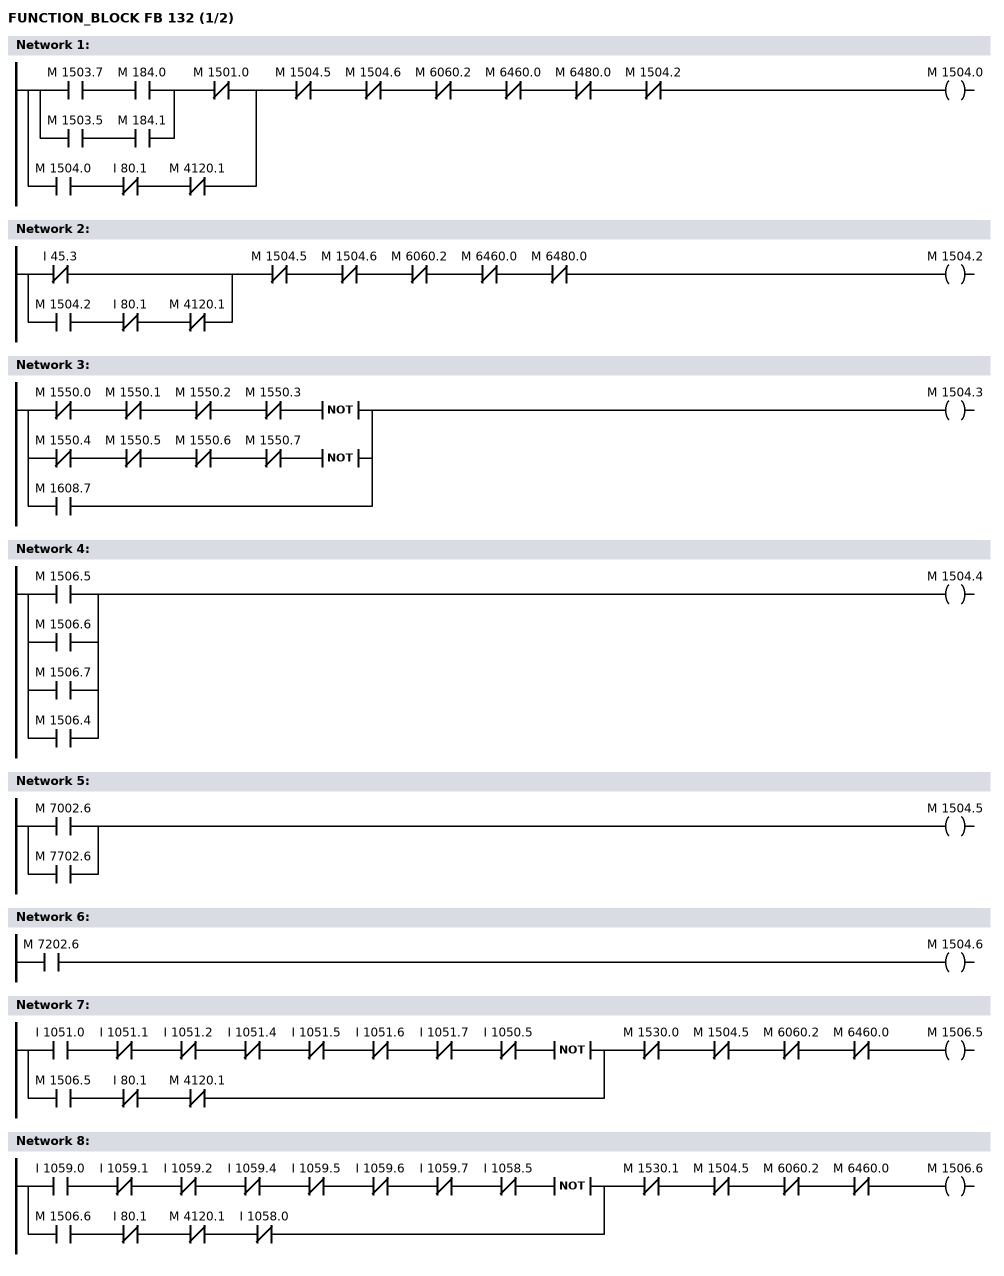

      A(    ;
      A(    ;
      A     M   1503.7;
      A     M    184.0;
      O     ;
      A     M   1503.5;
      A     M    184.1;
      )     ;
      AN    M   1501.0;
      O     ;
      A     M   1504.0;
      AN    I     80.1;
      AN    M   4120.1;
      )     ;
      AN    M   1504.5;
      AN    M   1504.6;
      AN    M   6060.2;
      AN    M   6460.0;
      AN    M   6480.0;
      AN    M   1504.2;
      =     M   1504.0;
NETWORK
TITLE =

      A(    ;
      ON    I     45.3;
      O     ;
      A     M   1504.2;
      AN    I     80.1;
      AN    M   4120.1;
      )     ;
      AN    M   1504.5;
      AN    M   1504.6;
      AN    M   6060.2;
      AN    M   6460.0;
      AN    M   6480.0;
      =     M   1504.2;
NETWORK
TITLE =

      AN    M   1550.0;
      AN    M   1550.1;
      AN    M   1550.2;
      AN    M   1550.3;
      NOT   ;
      O(    ;
      AN    M   1550.4;
      AN    M   1550.5;
      AN    M   1550.6;
      AN    M   1550.7;
      NOT   ;
      )     ;
      O     M   1608.7;
      =     M   1504.3;
NETWORK
TITLE =

      O     M   1506.5;
      O     M   1506.6;
      O     M   1506.7;
      O     M   1506.4;
      =     M   1504.4;
NETWORK
TITLE =

      O     M   7002.6;
      O     M   7702.6;
      =     M   1504.5;
NETWORK
TITLE =

      A     M   7202.6;
      =     M   1504.6;
NETWORK
TITLE =

      A(    ;
      A     I   1051.0;
      AN    I   1051.1;
      AN    I   1051.2;
      AN    I   1051.4;
      AN    I   1051.5;
      AN    I   1051.6;
      AN    I   1051.7;
      AN    I   1050.5;
      NOT   ;
      O     ;
      A     M   1506.5;
      AN    I     80.1;
      AN    M   4120.1;
      )     ;
      AN    M   1530.0;
      AN    M   1504.5;
      AN    M   6060.2;
      AN    M   6460.0;
      =     M   1506.5;
NETWORK
TITLE =

      A(    ;
      A     I   1059.0;
      AN    I   1059.1;
      AN    I   1059.2;
      AN    I   1059.4;
      AN    I   1059.5;
      AN    I   1059.6;
      AN    I   1059.7;
      AN    I   1058.5;
      NOT   ;
      O     ;
      A     M   1506.6;
      AN    I     80.1;
      AN    M   4120.1;
      AN    I   1058.0;
      )     ;
      AN    M   1530.1;
      AN    M   1504.5;
      AN    M   6060.2;
      AN    M   6460.0;
      =     M   1506.6;
NETWORK
TITLE =
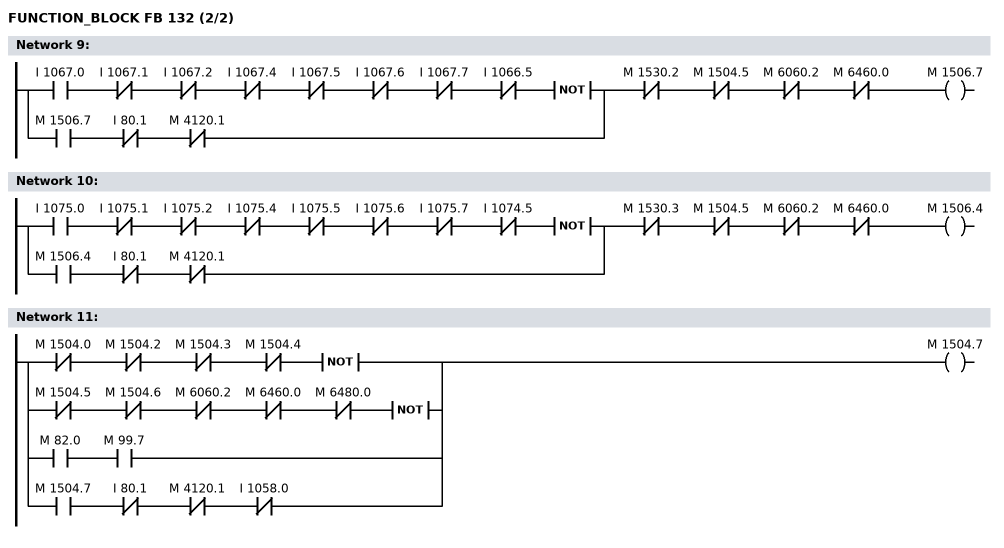

      A(    ;
      A     I   1067.0;
      AN    I   1067.1;
      AN    I   1067.2;
      AN    I   1067.4;
      AN    I   1067.5;
      AN    I   1067.6;
      AN    I   1067.7;
      AN    I   1066.5;
      NOT   ;
      O     ;
      A     M   1506.7;
      AN    I     80.1;
      AN    M   4120.1;
      )     ;
      AN    M   1530.2;
      AN    M   1504.5;
      AN    M   6060.2;
      AN    M   6460.0;
      =     M   1506.7;
NETWORK
TITLE =

      A(    ;
      A     I   1075.0;
      AN    I   1075.1;
      AN    I   1075.2;
      AN    I   1075.4;
      AN    I   1075.5;
      AN    I   1075.6;
      AN    I   1075.7;
      AN    I   1074.5;
      NOT   ;
      O     ;
      A     M   1506.4;
      AN    I     80.1;
      AN    M   4120.1;
      )     ;
      AN    M   1530.3;
      AN    M   1504.5;
      AN    M   6060.2;
      AN    M   6460.0;
      =     M   1506.4;
NETWORK
TITLE =

      AN    M   1504.0;
      AN    M   1504.2;
      AN    M   1504.3;
      AN    M   1504.4;
      NOT   ;
      O(    ;
      AN    M   1504.5;
      AN    M   1504.6;
      AN    M   6060.2;
      AN    M   6460.0;
      AN    M   6480.0;
      NOT   ;
      )     ;
      O     ;
      A     M     82.0;
      A     M     99.7;
      O     ;
      A     M   1504.7;
      AN    I     80.1;
      AN    M   4120.1;
      AN    I   1058.0;
      =     M   1504.7;
END_FUNCTION_BLOCK

DATA_BLOCK DB 132
TITLE =
VERSION : 0.0

 FB 132
BEGIN
END_DATA_BLOCK

FUNCTION FC 132 : VOID
TITLE =
VERSION : 0.1

BEGIN
NETWORK
TITLE =
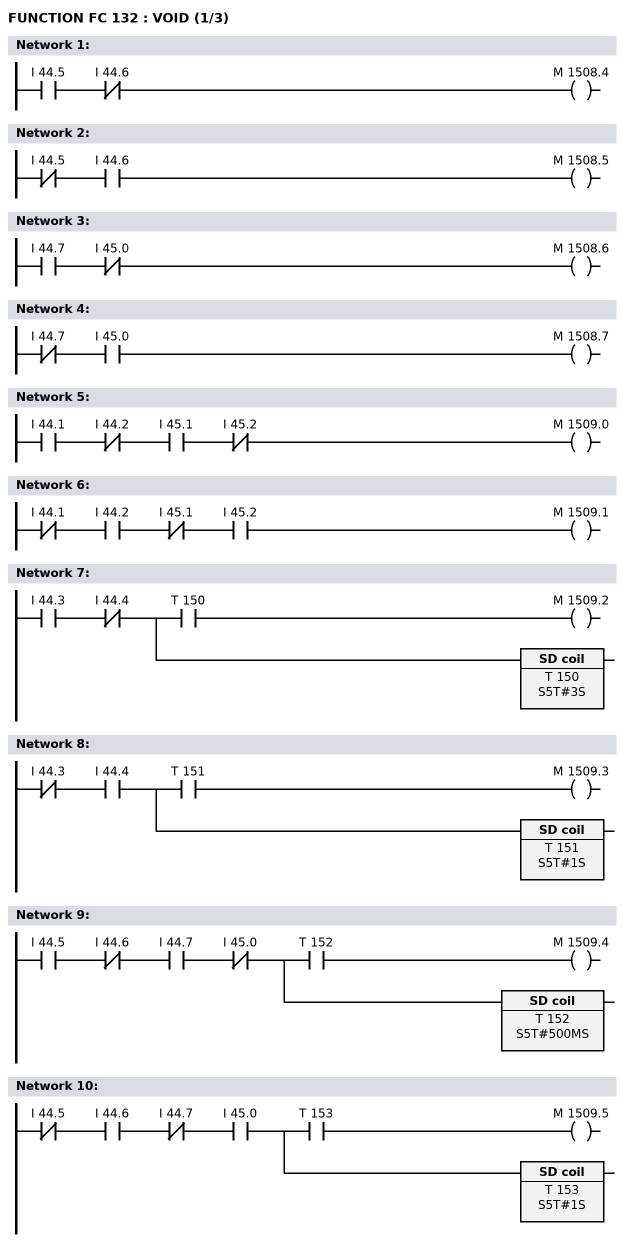

      A     I     44.5;
      AN    I     44.6;
      =     M   1508.4;
NETWORK
TITLE =

      AN    I     44.5;
      A     I     44.6;
      =     M   1508.5;
NETWORK
TITLE =

      A     I     44.7;
      AN    I     45.0;
      =     M   1508.6;
NETWORK
TITLE =

      AN    I     44.7;
      A     I     45.0;
      =     M   1508.7;
NETWORK
TITLE =

      A     I     44.1;
      AN    I     44.2;
      A     I     45.1;
      AN    I     45.2;
      =     M   1509.0;
NETWORK
TITLE =

      AN    I     44.1;
      A     I     44.2;
      AN    I     45.1;
      A     I     45.2;
      =     M   1509.1;
NETWORK
TITLE =

      A     I     44.3;
      AN    I     44.4;
      =     L      0.0;
      A     L      0.0;
      A     T    150;
      =     M   1509.2;
      A     L      0.0;
      BLD   102;
      L     S5T#3S;
      SD    T    150;
NETWORK
TITLE =

      AN    I     44.3;
      A     I     44.4;
      =     L      0.0;
      A     L      0.0;
      A     T    151;
      =     M   1509.3;
      A     L      0.0;
      BLD   102;
      L     S5T#1S;
      SD    T    151;
NETWORK
TITLE =

      A     I     44.5;
      AN    I     44.6;
      A     I     44.7;
      AN    I     45.0;
      =     L      0.0;
      A     L      0.0;
      A     T    152;
      =     M   1509.4;
      A     L      0.0;
      BLD   102;
      L     S5T#500MS;
      SD    T    152;
NETWORK
TITLE =

      AN    I     44.5;
      A     I     44.6;
      AN    I     44.7;
      A     I     45.0;
      =     L      0.0;
      A     L      0.0;
      A     T    153;
      =     M   1509.5;
      A     L      0.0;
      BLD   102;
      L     S5T#1S;
      SD    T    153;
NETWORK
TITLE =
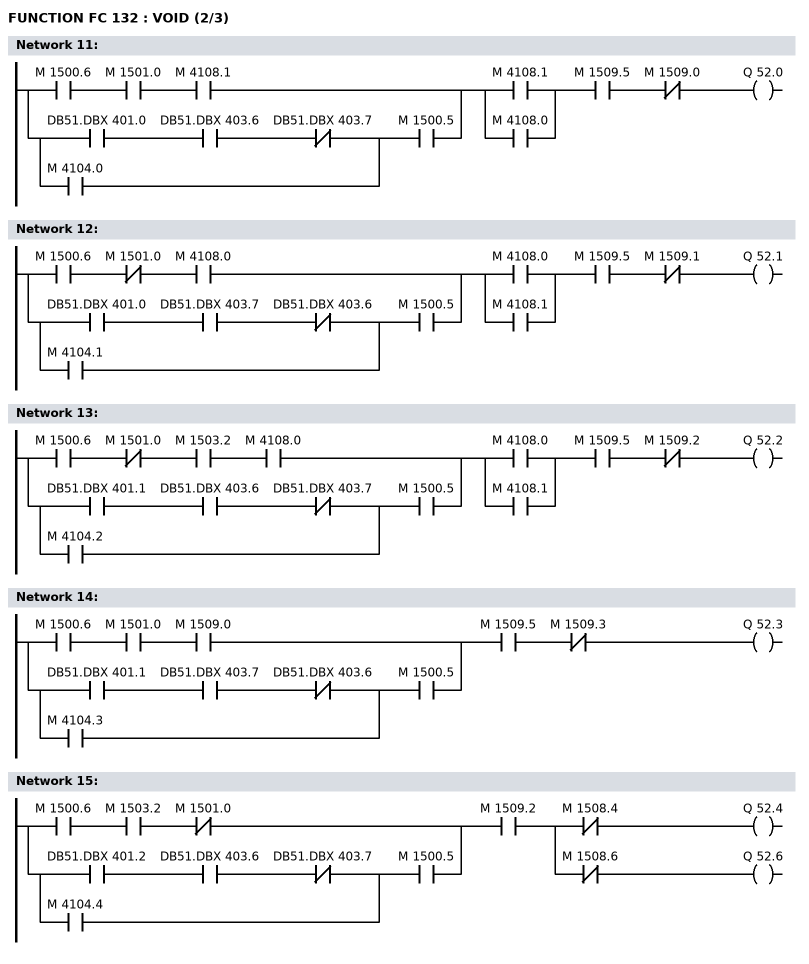

      A(    ;
      A     M   1500.6;
      A     M   1501.0;
      A     M   4108.1;
      O     ;
      A(    ;
      A     DB51.DBX  401.0;
      A     DB51.DBX  403.6;
      AN    DB51.DBX  403.7;
      O     M   4104.0;
      )     ;
      A     M   1500.5;
      )     ;
      A(    ;
      O     M   4108.1;
      O     M   4108.0;
      )     ;
      A     M   1509.5;
      AN    M   1509.0;
      =     Q     52.0;
NETWORK
TITLE =

      A(    ;
      A     M   1500.6;
      AN    M   1501.0;
      A     M   4108.0;
      O     ;
      A(    ;
      A     DB51.DBX  401.0;
      A     DB51.DBX  403.7;
      AN    DB51.DBX  403.6;
      O     M   4104.1;
      )     ;
      A     M   1500.5;
      )     ;
      A(    ;
      O     M   4108.0;
      O     M   4108.1;
      )     ;
      A     M   1509.5;
      AN    M   1509.1;
      =     Q     52.1;
NETWORK
TITLE =

      A(    ;
      A     M   1500.6;
      AN    M   1501.0;
      A     M   1503.2;
      A     M   4108.0;
      O     ;
      A(    ;
      A     DB51.DBX  401.1;
      A     DB51.DBX  403.6;
      AN    DB51.DBX  403.7;
      O     M   4104.2;
      )     ;
      A     M   1500.5;
      )     ;
      A(    ;
      O     M   4108.0;
      O     M   4108.1;
      )     ;
      A     M   1509.5;
      AN    M   1509.2;
      =     Q     52.2;
NETWORK
TITLE =

      A(    ;
      A     M   1500.6;
      A     M   1501.0;
      A     M   1509.0;
      O     ;
      A(    ;
      A     DB51.DBX  401.1;
      A     DB51.DBX  403.7;
      AN    DB51.DBX  403.6;
      O     M   4104.3;
      )     ;
      A     M   1500.5;
      )     ;
      A     M   1509.5;
      AN    M   1509.3;
      =     Q     52.3;
NETWORK
TITLE =

      A(    ;
      A     M   1500.6;
      A     M   1503.2;
      AN    M   1501.0;
      O     ;
      A(    ;
      A     DB51.DBX  401.2;
      A     DB51.DBX  403.6;
      AN    DB51.DBX  403.7;
      O     M   4104.4;
      )     ;
      A     M   1500.5;
      )     ;
      A     M   1509.2;
      =     L      0.0;
      A     L      0.0;
      AN    M   1508.4;
      =     Q     52.4;
      A     L      0.0;
      AN    M   1508.6;
      =     Q     52.6;
NETWORK
TITLE =
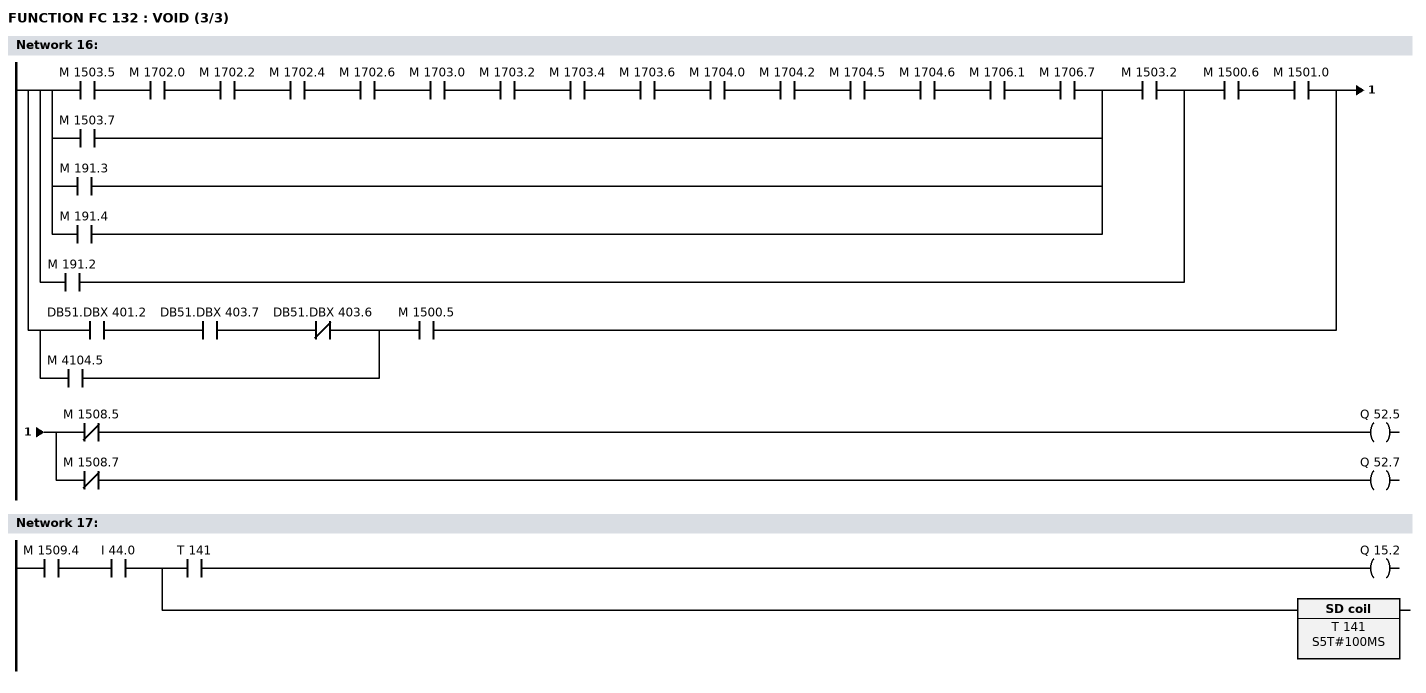

      A(    ;
      A(    ;
      A     M   1503.5;
      A     M   1702.0;
      A     M   1702.2;
      A     M   1702.4;
      A     M   1702.6;
      A     M   1703.0;
      A     M   1703.2;
      A     M   1703.4;
      A     M   1703.6;
      A     M   1704.0;
      A     M   1704.2;
      A     M   1704.5;
      A     M   1704.6;
      A     M   1706.1;
      A     M   1706.7;
      O     M   1503.7;
      O     M    191.3;
      O     M    191.4;
      )     ;
      A     M   1503.2;
      O     M    191.2;
      )     ;
      A     M   1500.6;
      A     M   1501.0;
      O     ;
      A(    ;
      A     DB51.DBX  401.2;
      A     DB51.DBX  403.7;
      AN    DB51.DBX  403.6;
      O     M   4104.5;
      )     ;
      A     M   1500.5;
      =     L      0.0;
      A     L      0.0;
      AN    M   1508.5;
      =     Q     52.5;
      A     L      0.0;
      AN    M   1508.7;
      =     Q     52.7;
NETWORK
TITLE =

      A     M   1509.4;
      A     I     44.0;
      =     L      0.0;
      A     L      0.0;
      A     T    141;
      =     Q     15.2;
      A     L      0.0;
      BLD   102;
      L     S5T#100MS;
      SD    T    141;
END_FUNCTION

FUNCTION_BLOCK FB 133
TITLE =
VERSION : 0.1


VAR
  S707_LM_DC_PIN : FB 424;
  S707_LM_DC_1ST_CLAMP1 : FB 424;
  S707_LM_DC_1ST_CLAMP2 : FB 424;
  S707_LM_DC_1ST_CLAMP3 : FB 424;
  S707_LM_DC_1ST_CLAMP4 : FB 424;
  S707_LM_DC_2ND_CLAMP1 : FB 424;
  S707_LM_DC_2ND_CLAMP2 : FB 424;
  S707_LM_DC_2ND_CLAMP3 : FB 424;
  S707_LM_DC_2ND_CLAMP4 : FB 424;
  S707_LM_DC_2ND_CLAMP5 : FB 424;
  S707_LM_DC_STK_PIN : FB 424;
  S707_LM_DC_OTR_CLAMP : FB 424;
  S707_LM_DC_ASSY_CLAMP : FB 424;
  S707_LM_DC_FF_PIN : FB 424;
  S707_LM_DC_FF_CLAMP : FB 424;
  S707_LM_DC_2ND_CLAMP6 : FB 424;
  S707_LM_DC_2ND_CLAMP7 : FB 424;
  S707_LM_DC_1ST_CLAMP5 : FB 424;
END_VAR
BEGIN
NETWORK
TITLE =
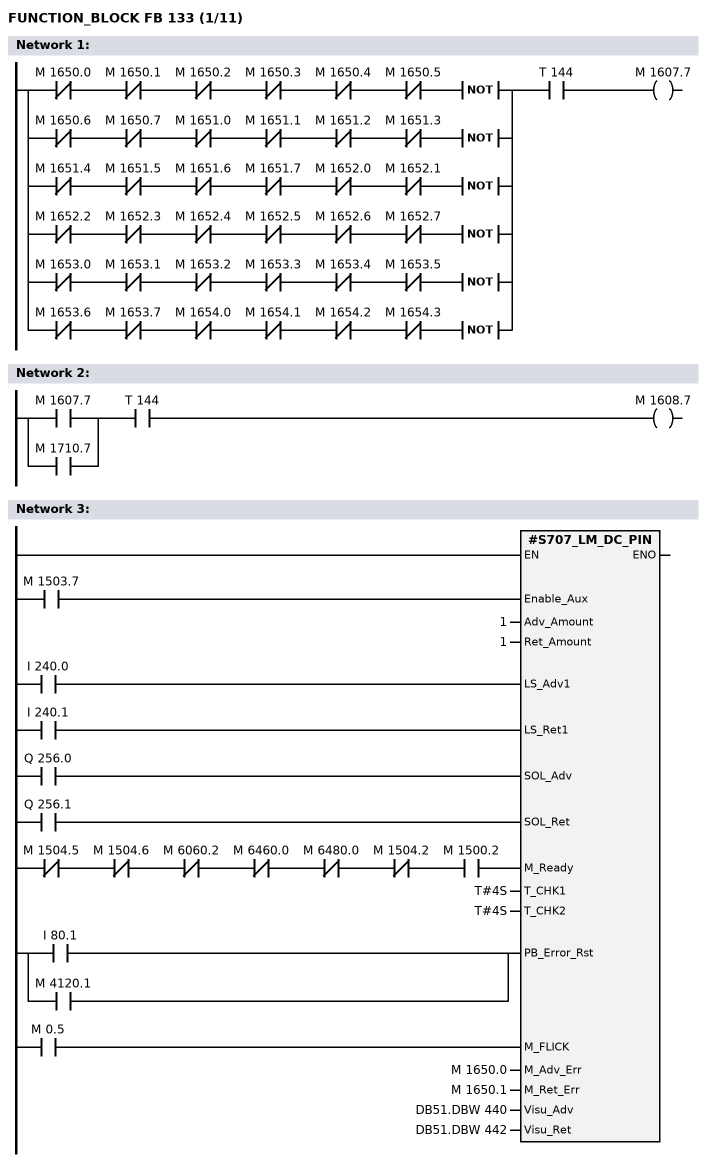

      A(    ;
      AN    M   1650.0;
      AN    M   1650.1;
      AN    M   1650.2;
      AN    M   1650.3;
      AN    M   1650.4;
      AN    M   1650.5;
      NOT   ;
      O(    ;
      AN    M   1650.6;
      AN    M   1650.7;
      AN    M   1651.0;
      AN    M   1651.1;
      AN    M   1651.2;
      AN    M   1651.3;
      NOT   ;
      )     ;
      O(    ;
      AN    M   1651.4;
      AN    M   1651.5;
      AN    M   1651.6;
      AN    M   1651.7;
      AN    M   1652.0;
      AN    M   1652.1;
      NOT   ;
      )     ;
      O(    ;
      AN    M   1652.2;
      AN    M   1652.3;
      AN    M   1652.4;
      AN    M   1652.5;
      AN    M   1652.6;
      AN    M   1652.7;
      NOT   ;
      )     ;
      O(    ;
      AN    M   1653.0;
      AN    M   1653.1;
      AN    M   1653.2;
      AN    M   1653.3;
      AN    M   1653.4;
      AN    M   1653.5;
      NOT   ;
      )     ;
      O(    ;
      AN    M   1653.6;
      AN    M   1653.7;
      AN    M   1654.0;
      AN    M   1654.1;
      AN    M   1654.2;
      AN    M   1654.3;
      NOT   ;
      )     ;
      )     ;
      A     T    144;
      =     M   1607.7;
NETWORK
TITLE =

      A(    ;
      O     M   1607.7;
      O     M   1710.7;
      )     ;
      A     T    144;
      =     M   1608.7;
NETWORK
TITLE =

      A     M   1503.7;
      =     L      0.0;
      BLD   103;
      A     I    240.0;
      =     L      0.1;
      BLD   103;
      A     I    240.1;
      =     L      0.2;
      BLD   103;
      A     Q    256.0;
      =     L      1.1;
      BLD   103;
      A     Q    256.1;
      =     L      1.2;
      BLD   103;
      AN    M   1504.5;
      AN    M   1504.6;
      AN    M   6060.2;
      AN    M   6460.0;
      AN    M   6480.0;
      AN    M   1504.2;
      A     M   1500.2;
      =     L      1.3;
      BLD   103;
      A(    ;
      O     I     80.1;
      O     M   4120.1;
      )     ;
      =     L      1.5;
      BLD   103;
      A     M      0.5;
      =     L      1.6;
      BLD   103;
      CALL #S707_LM_DC_PIN (
           Enable_Aux               := L      0.0,
           Adv_Amount               := 1,
           Ret_Amount               := 1,
           LS_Adv1                  := L      0.1,
           LS_Ret1                  := L      0.2,
           SOL_Adv                  := L      1.1,
           SOL_Ret                  := L      1.2,
           M_Ready                  := L      1.3,
           T_CHK1                   := T#4S,
           T_CHK2                   := T#4S,
           PB_Error_Rst             := L      1.5,
           M_FLICK                  := L      1.6,
           M_Adv_Err                := M   1650.0,
           M_Ret_Err                := M   1650.1,
           Visu_Adv                 := DB51.DBW  440,
           Visu_Ret                 := DB51.DBW  442);
      NOP   0;
NETWORK
TITLE =
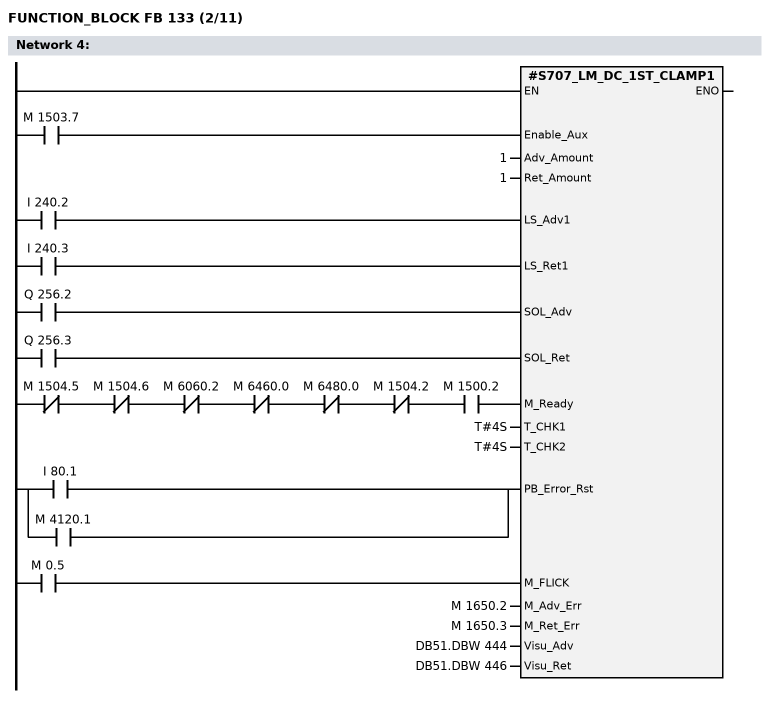

      A     M   1503.7;
      =     L      0.0;
      BLD   103;
      A     I    240.2;
      =     L      0.1;
      BLD   103;
      A     I    240.3;
      =     L      0.2;
      BLD   103;
      A     Q    256.2;
      =     L      1.1;
      BLD   103;
      A     Q    256.3;
      =     L      1.2;
      BLD   103;
      AN    M   1504.5;
      AN    M   1504.6;
      AN    M   6060.2;
      AN    M   6460.0;
      AN    M   6480.0;
      AN    M   1504.2;
      A     M   1500.2;
      =     L      1.3;
      BLD   103;
      A(    ;
      O     I     80.1;
      O     M   4120.1;
      )     ;
      =     L      1.5;
      BLD   103;
      A     M      0.5;
      =     L      1.6;
      BLD   103;
      CALL #S707_LM_DC_1ST_CLAMP1 (
           Enable_Aux               := L      0.0,
           Adv_Amount               := 1,
           Ret_Amount               := 1,
           LS_Adv1                  := L      0.1,
           LS_Ret1                  := L      0.2,
           SOL_Adv                  := L      1.1,
           SOL_Ret                  := L      1.2,
           M_Ready                  := L      1.3,
           T_CHK1                   := T#4S,
           T_CHK2                   := T#4S,
           PB_Error_Rst             := L      1.5,
           M_FLICK                  := L      1.6,
           M_Adv_Err                := M   1650.2,
           M_Ret_Err                := M   1650.3,
           Visu_Adv                 := DB51.DBW  444,
           Visu_Ret                 := DB51.DBW  446);
      NOP   0;
NETWORK
TITLE =
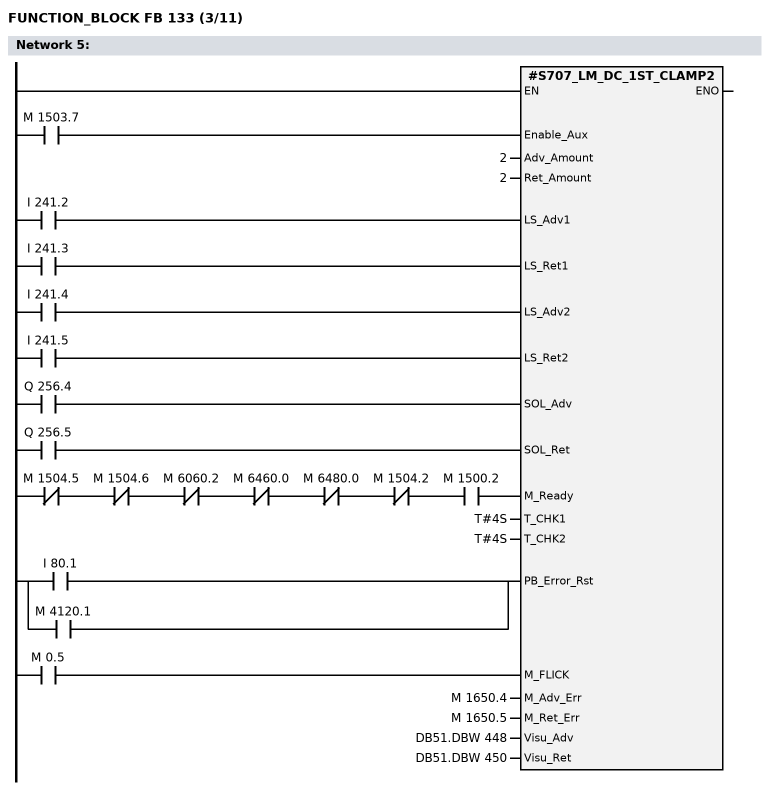

      A     M   1503.7;
      =     L      0.0;
      BLD   103;
      A     I    241.2;
      =     L      0.1;
      BLD   103;
      A     I    241.3;
      =     L      0.2;
      BLD   103;
      A     I    241.4;
      =     L      0.3;
      BLD   103;
      A     I    241.5;
      =     L      0.4;
      BLD   103;
      A     Q    256.4;
      =     L      1.1;
      BLD   103;
      A     Q    256.5;
      =     L      1.2;
      BLD   103;
      AN    M   1504.5;
      AN    M   1504.6;
      AN    M   6060.2;
      AN    M   6460.0;
      AN    M   6480.0;
      AN    M   1504.2;
      A     M   1500.2;
      =     L      1.3;
      BLD   103;
      A(    ;
      O     I     80.1;
      O     M   4120.1;
      )     ;
      =     L      1.5;
      BLD   103;
      A     M      0.5;
      =     L      1.6;
      BLD   103;
      CALL #S707_LM_DC_1ST_CLAMP2 (
           Enable_Aux               := L      0.0,
           Adv_Amount               := 2,
           Ret_Amount               := 2,
           LS_Adv1                  := L      0.1,
           LS_Ret1                  := L      0.2,
           LS_Adv2                  := L      0.3,
           LS_Ret2                  := L      0.4,
           SOL_Adv                  := L      1.1,
           SOL_Ret                  := L      1.2,
           M_Ready                  := L      1.3,
           T_CHK1                   := T#4S,
           T_CHK2                   := T#4S,
           PB_Error_Rst             := L      1.5,
           M_FLICK                  := L      1.6,
           M_Adv_Err                := M   1650.4,
           M_Ret_Err                := M   1650.5,
           Visu_Adv                 := DB51.DBW  448,
           Visu_Ret                 := DB51.DBW  450);
      NOP   0;
NETWORK
TITLE =
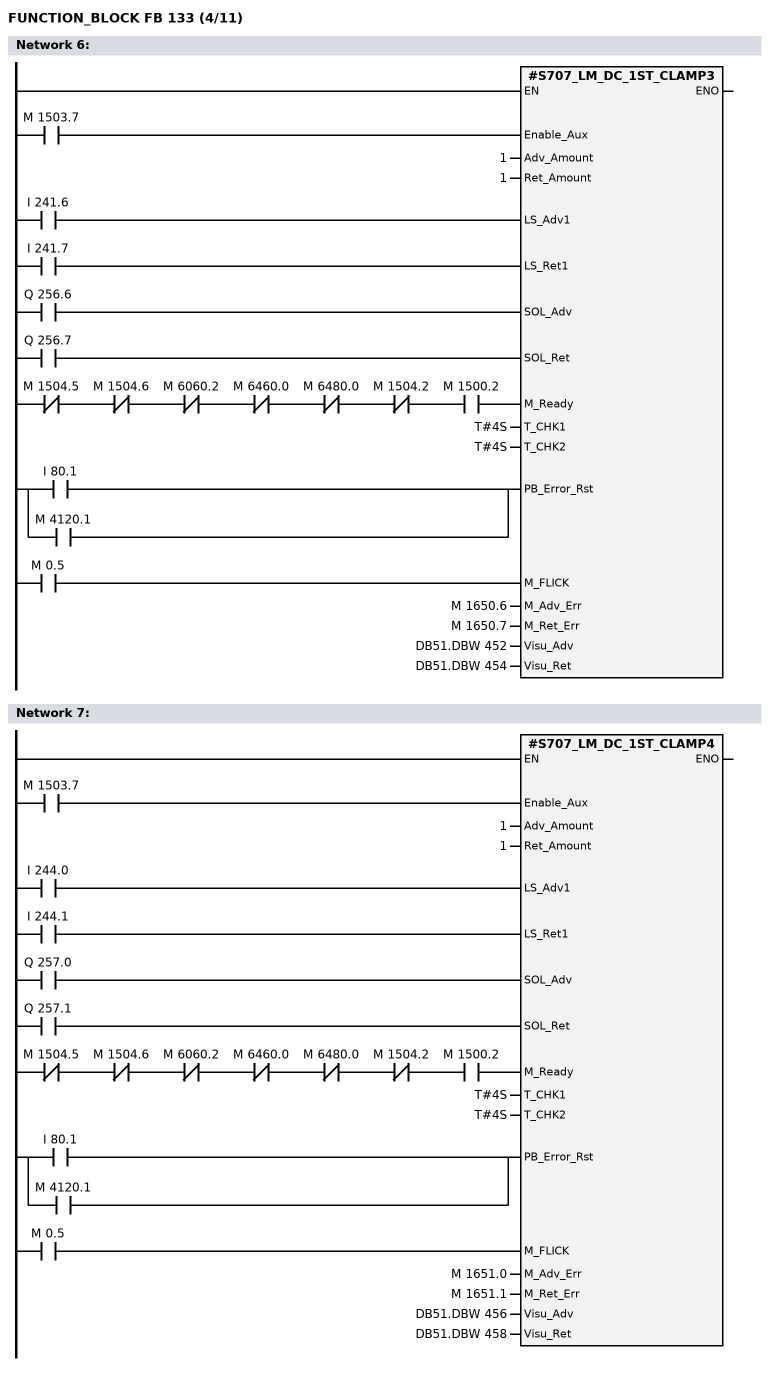

      A     M   1503.7;
      =     L      0.0;
      BLD   103;
      A     I    241.6;
      =     L      0.1;
      BLD   103;
      A     I    241.7;
      =     L      0.2;
      BLD   103;
      A     Q    256.6;
      =     L      1.1;
      BLD   103;
      A     Q    256.7;
      =     L      1.2;
      BLD   103;
      AN    M   1504.5;
      AN    M   1504.6;
      AN    M   6060.2;
      AN    M   6460.0;
      AN    M   6480.0;
      AN    M   1504.2;
      A     M   1500.2;
      =     L      1.3;
      BLD   103;
      A(    ;
      O     I     80.1;
      O     M   4120.1;
      )     ;
      =     L      1.5;
      BLD   103;
      A     M      0.5;
      =     L      1.6;
      BLD   103;
      CALL #S707_LM_DC_1ST_CLAMP3 (
           Enable_Aux               := L      0.0,
           Adv_Amount               := 1,
           Ret_Amount               := 1,
           LS_Adv1                  := L      0.1,
           LS_Ret1                  := L      0.2,
           SOL_Adv                  := L      1.1,
           SOL_Ret                  := L      1.2,
           M_Ready                  := L      1.3,
           T_CHK1                   := T#4S,
           T_CHK2                   := T#4S,
           PB_Error_Rst             := L      1.5,
           M_FLICK                  := L      1.6,
           M_Adv_Err                := M   1650.6,
           M_Ret_Err                := M   1650.7,
           Visu_Adv                 := DB51.DBW  452,
           Visu_Ret                 := DB51.DBW  454);
      NOP   0;
NETWORK
TITLE =

      A     M   1503.7;
      =     L      0.0;
      BLD   103;
      A     I    244.0;
      =     L      0.1;
      BLD   103;
      A     I    244.1;
      =     L      0.2;
      BLD   103;
      A     Q    257.0;
      =     L      1.1;
      BLD   103;
      A     Q    257.1;
      =     L      1.2;
      BLD   103;
      AN    M   1504.5;
      AN    M   1504.6;
      AN    M   6060.2;
      AN    M   6460.0;
      AN    M   6480.0;
      AN    M   1504.2;
      A     M   1500.2;
      =     L      1.3;
      BLD   103;
      A(    ;
      O     I     80.1;
      O     M   4120.1;
      )     ;
      =     L      1.5;
      BLD   103;
      A     M      0.5;
      =     L      1.6;
      BLD   103;
      CALL #S707_LM_DC_1ST_CLAMP4 (
           Enable_Aux               := L      0.0,
           Adv_Amount               := 1,
           Ret_Amount               := 1,
           LS_Adv1                  := L      0.1,
           LS_Ret1                  := L      0.2,
           SOL_Adv                  := L      1.1,
           SOL_Ret                  := L      1.2,
           M_Ready                  := L      1.3,
           T_CHK1                   := T#4S,
           T_CHK2                   := T#4S,
           PB_Error_Rst             := L      1.5,
           M_FLICK                  := L      1.6,
           M_Adv_Err                := M   1651.0,
           M_Ret_Err                := M   1651.1,
           Visu_Adv                 := DB51.DBW  456,
           Visu_Ret                 := DB51.DBW  458);
      NOP   0;
NETWORK
TITLE =
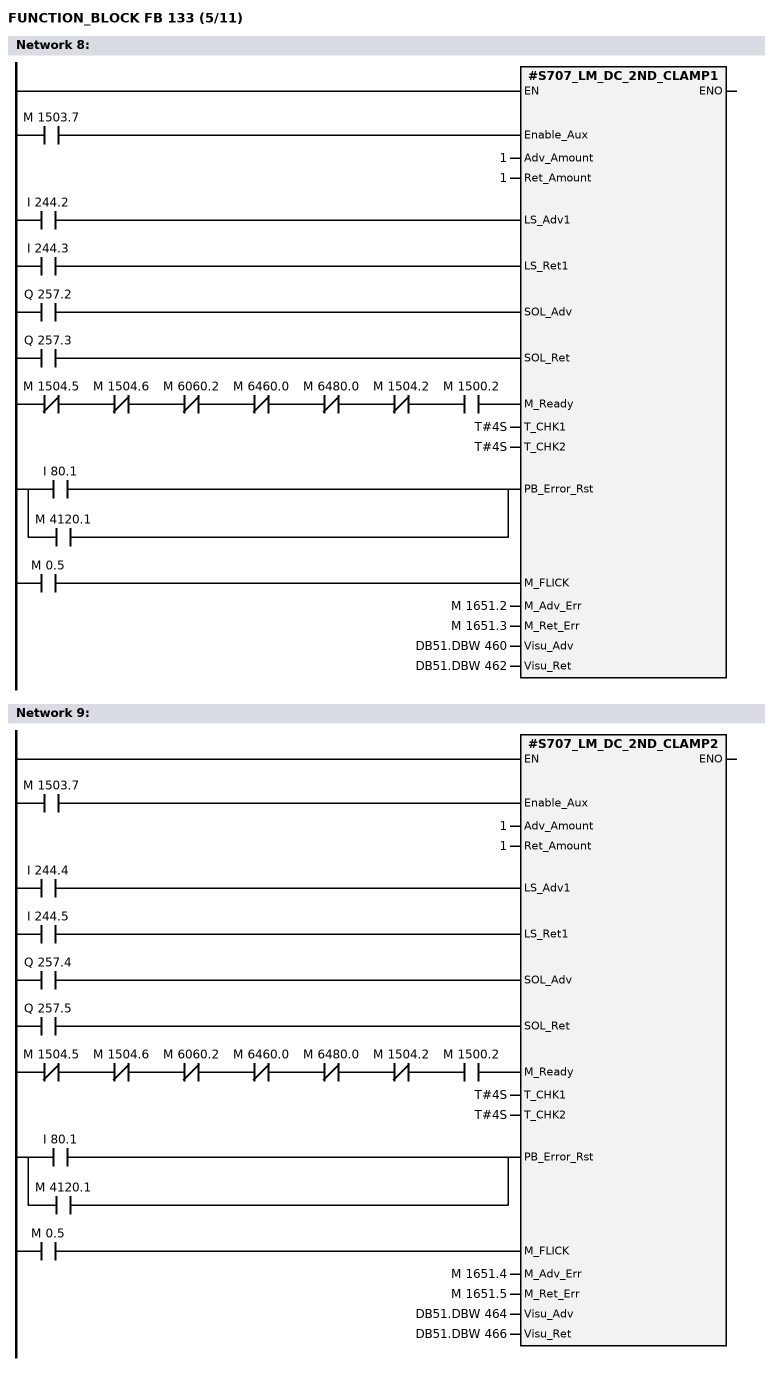

      A     M   1503.7;
      =     L      0.0;
      BLD   103;
      A     I    244.2;
      =     L      0.1;
      BLD   103;
      A     I    244.3;
      =     L      0.2;
      BLD   103;
      A     Q    257.2;
      =     L      1.1;
      BLD   103;
      A     Q    257.3;
      =     L      1.2;
      BLD   103;
      AN    M   1504.5;
      AN    M   1504.6;
      AN    M   6060.2;
      AN    M   6460.0;
      AN    M   6480.0;
      AN    M   1504.2;
      A     M   1500.2;
      =     L      1.3;
      BLD   103;
      A(    ;
      O     I     80.1;
      O     M   4120.1;
      )     ;
      =     L      1.5;
      BLD   103;
      A     M      0.5;
      =     L      1.6;
      BLD   103;
      CALL #S707_LM_DC_2ND_CLAMP1 (
           Enable_Aux               := L      0.0,
           Adv_Amount               := 1,
           Ret_Amount               := 1,
           LS_Adv1                  := L      0.1,
           LS_Ret1                  := L      0.2,
           SOL_Adv                  := L      1.1,
           SOL_Ret                  := L      1.2,
           M_Ready                  := L      1.3,
           T_CHK1                   := T#4S,
           T_CHK2                   := T#4S,
           PB_Error_Rst             := L      1.5,
           M_FLICK                  := L      1.6,
           M_Adv_Err                := M   1651.2,
           M_Ret_Err                := M   1651.3,
           Visu_Adv                 := DB51.DBW  460,
           Visu_Ret                 := DB51.DBW  462);
      NOP   0;
NETWORK
TITLE =

      A     M   1503.7;
      =     L      0.0;
      BLD   103;
      A     I    244.4;
      =     L      0.1;
      BLD   103;
      A     I    244.5;
      =     L      0.2;
      BLD   103;
      A     Q    257.4;
      =     L      1.1;
      BLD   103;
      A     Q    257.5;
      =     L      1.2;
      BLD   103;
      AN    M   1504.5;
      AN    M   1504.6;
      AN    M   6060.2;
      AN    M   6460.0;
      AN    M   6480.0;
      AN    M   1504.2;
      A     M   1500.2;
      =     L      1.3;
      BLD   103;
      A(    ;
      O     I     80.1;
      O     M   4120.1;
      )     ;
      =     L      1.5;
      BLD   103;
      A     M      0.5;
      =     L      1.6;
      BLD   103;
      CALL #S707_LM_DC_2ND_CLAMP2 (
           Enable_Aux               := L      0.0,
           Adv_Amount               := 1,
           Ret_Amount               := 1,
           LS_Adv1                  := L      0.1,
           LS_Ret1                  := L      0.2,
           SOL_Adv                  := L      1.1,
           SOL_Ret                  := L      1.2,
           M_Ready                  := L      1.3,
           T_CHK1                   := T#4S,
           T_CHK2                   := T#4S,
           PB_Error_Rst             := L      1.5,
           M_FLICK                  := L      1.6,
           M_Adv_Err                := M   1651.4,
           M_Ret_Err                := M   1651.5,
           Visu_Adv                 := DB51.DBW  464,
           Visu_Ret                 := DB51.DBW  466);
      NOP   0;
NETWORK
TITLE =
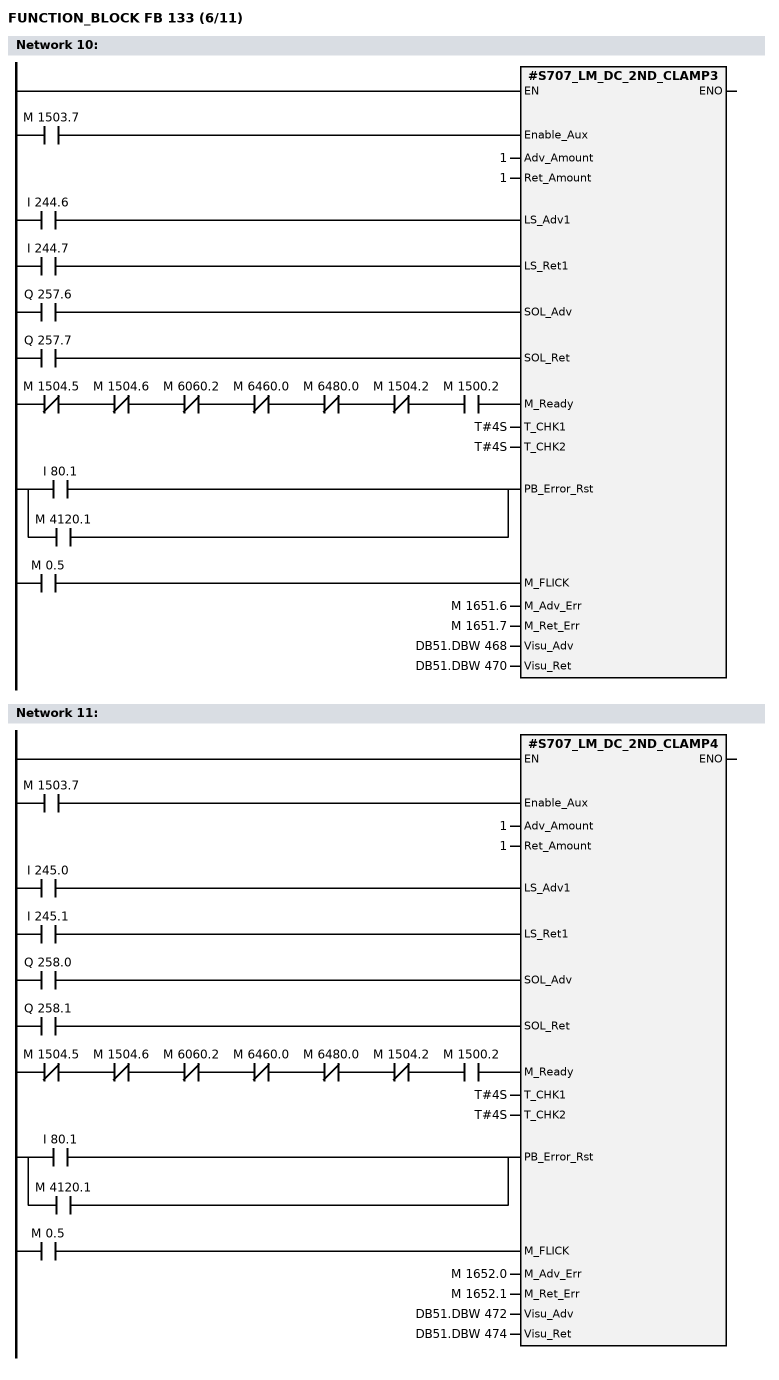

      A     M   1503.7;
      =     L      0.0;
      BLD   103;
      A     I    244.6;
      =     L      0.1;
      BLD   103;
      A     I    244.7;
      =     L      0.2;
      BLD   103;
      A     Q    257.6;
      =     L      1.1;
      BLD   103;
      A     Q    257.7;
      =     L      1.2;
      BLD   103;
      AN    M   1504.5;
      AN    M   1504.6;
      AN    M   6060.2;
      AN    M   6460.0;
      AN    M   6480.0;
      AN    M   1504.2;
      A     M   1500.2;
      =     L      1.3;
      BLD   103;
      A(    ;
      O     I     80.1;
      O     M   4120.1;
      )     ;
      =     L      1.5;
      BLD   103;
      A     M      0.5;
      =     L      1.6;
      BLD   103;
      CALL #S707_LM_DC_2ND_CLAMP3 (
           Enable_Aux               := L      0.0,
           Adv_Amount               := 1,
           Ret_Amount               := 1,
           LS_Adv1                  := L      0.1,
           LS_Ret1                  := L      0.2,
           SOL_Adv                  := L      1.1,
           SOL_Ret                  := L      1.2,
           M_Ready                  := L      1.3,
           T_CHK1                   := T#4S,
           T_CHK2                   := T#4S,
           PB_Error_Rst             := L      1.5,
           M_FLICK                  := L      1.6,
           M_Adv_Err                := M   1651.6,
           M_Ret_Err                := M   1651.7,
           Visu_Adv                 := DB51.DBW  468,
           Visu_Ret                 := DB51.DBW  470);
      NOP   0;
NETWORK
TITLE =

      A     M   1503.7;
      =     L      0.0;
      BLD   103;
      A     I    245.0;
      =     L      0.1;
      BLD   103;
      A     I    245.1;
      =     L      0.2;
      BLD   103;
      A     Q    258.0;
      =     L      1.1;
      BLD   103;
      A     Q    258.1;
      =     L      1.2;
      BLD   103;
      AN    M   1504.5;
      AN    M   1504.6;
      AN    M   6060.2;
      AN    M   6460.0;
      AN    M   6480.0;
      AN    M   1504.2;
      A     M   1500.2;
      =     L      1.3;
      BLD   103;
      A(    ;
      O     I     80.1;
      O     M   4120.1;
      )     ;
      =     L      1.5;
      BLD   103;
      A     M      0.5;
      =     L      1.6;
      BLD   103;
      CALL #S707_LM_DC_2ND_CLAMP4 (
           Enable_Aux               := L      0.0,
           Adv_Amount               := 1,
           Ret_Amount               := 1,
           LS_Adv1                  := L      0.1,
           LS_Ret1                  := L      0.2,
           SOL_Adv                  := L      1.1,
           SOL_Ret                  := L      1.2,
           M_Ready                  := L      1.3,
           T_CHK1                   := T#4S,
           T_CHK2                   := T#4S,
           PB_Error_Rst             := L      1.5,
           M_FLICK                  := L      1.6,
           M_Adv_Err                := M   1652.0,
           M_Ret_Err                := M   1652.1,
           Visu_Adv                 := DB51.DBW  472,
           Visu_Ret                 := DB51.DBW  474);
      NOP   0;
NETWORK
TITLE =
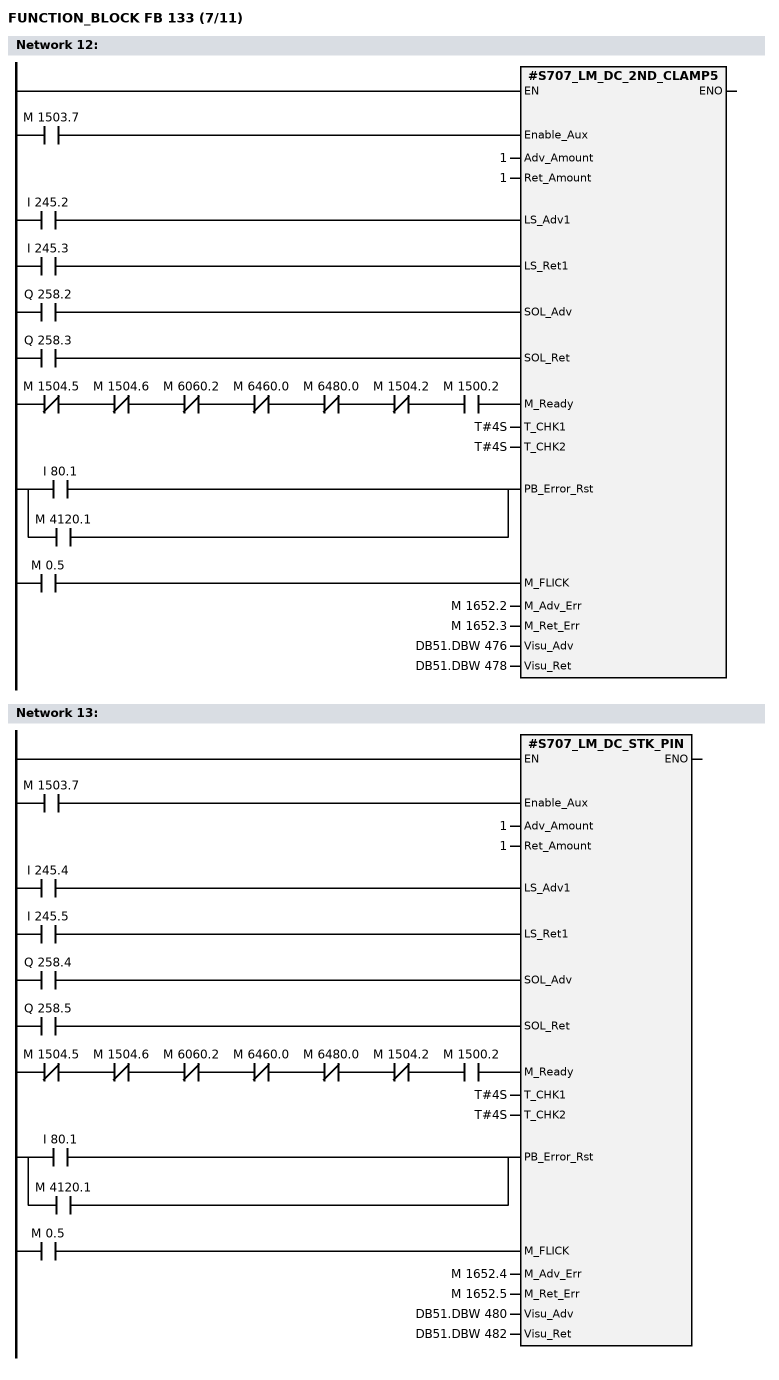

      A     M   1503.7;
      =     L      0.0;
      BLD   103;
      A     I    245.2;
      =     L      0.1;
      BLD   103;
      A     I    245.3;
      =     L      0.2;
      BLD   103;
      A     Q    258.2;
      =     L      1.1;
      BLD   103;
      A     Q    258.3;
      =     L      1.2;
      BLD   103;
      AN    M   1504.5;
      AN    M   1504.6;
      AN    M   6060.2;
      AN    M   6460.0;
      AN    M   6480.0;
      AN    M   1504.2;
      A     M   1500.2;
      =     L      1.3;
      BLD   103;
      A(    ;
      O     I     80.1;
      O     M   4120.1;
      )     ;
      =     L      1.5;
      BLD   103;
      A     M      0.5;
      =     L      1.6;
      BLD   103;
      CALL #S707_LM_DC_2ND_CLAMP5 (
           Enable_Aux               := L      0.0,
           Adv_Amount               := 1,
           Ret_Amount               := 1,
           LS_Adv1                  := L      0.1,
           LS_Ret1                  := L      0.2,
           SOL_Adv                  := L      1.1,
           SOL_Ret                  := L      1.2,
           M_Ready                  := L      1.3,
           T_CHK1                   := T#4S,
           T_CHK2                   := T#4S,
           PB_Error_Rst             := L      1.5,
           M_FLICK                  := L      1.6,
           M_Adv_Err                := M   1652.2,
           M_Ret_Err                := M   1652.3,
           Visu_Adv                 := DB51.DBW  476,
           Visu_Ret                 := DB51.DBW  478);
      NOP   0;
NETWORK
TITLE =

      A     M   1503.7;
      =     L      0.0;
      BLD   103;
      A     I    245.4;
      =     L      0.1;
      BLD   103;
      A     I    245.5;
      =     L      0.2;
      BLD   103;
      A     Q    258.4;
      =     L      1.1;
      BLD   103;
      A     Q    258.5;
      =     L      1.2;
      BLD   103;
      AN    M   1504.5;
      AN    M   1504.6;
      AN    M   6060.2;
      AN    M   6460.0;
      AN    M   6480.0;
      AN    M   1504.2;
      A     M   1500.2;
      =     L      1.3;
      BLD   103;
      A(    ;
      O     I     80.1;
      O     M   4120.1;
      )     ;
      =     L      1.5;
      BLD   103;
      A     M      0.5;
      =     L      1.6;
      BLD   103;
      CALL #S707_LM_DC_STK_PIN (
           Enable_Aux               := L      0.0,
           Adv_Amount               := 1,
           Ret_Amount               := 1,
           LS_Adv1                  := L      0.1,
           LS_Ret1                  := L      0.2,
           SOL_Adv                  := L      1.1,
           SOL_Ret                  := L      1.2,
           M_Ready                  := L      1.3,
           T_CHK1                   := T#4S,
           T_CHK2                   := T#4S,
           PB_Error_Rst             := L      1.5,
           M_FLICK                  := L      1.6,
           M_Adv_Err                := M   1652.4,
           M_Ret_Err                := M   1652.5,
           Visu_Adv                 := DB51.DBW  480,
           Visu_Ret                 := DB51.DBW  482);
      NOP   0;
NETWORK
TITLE =
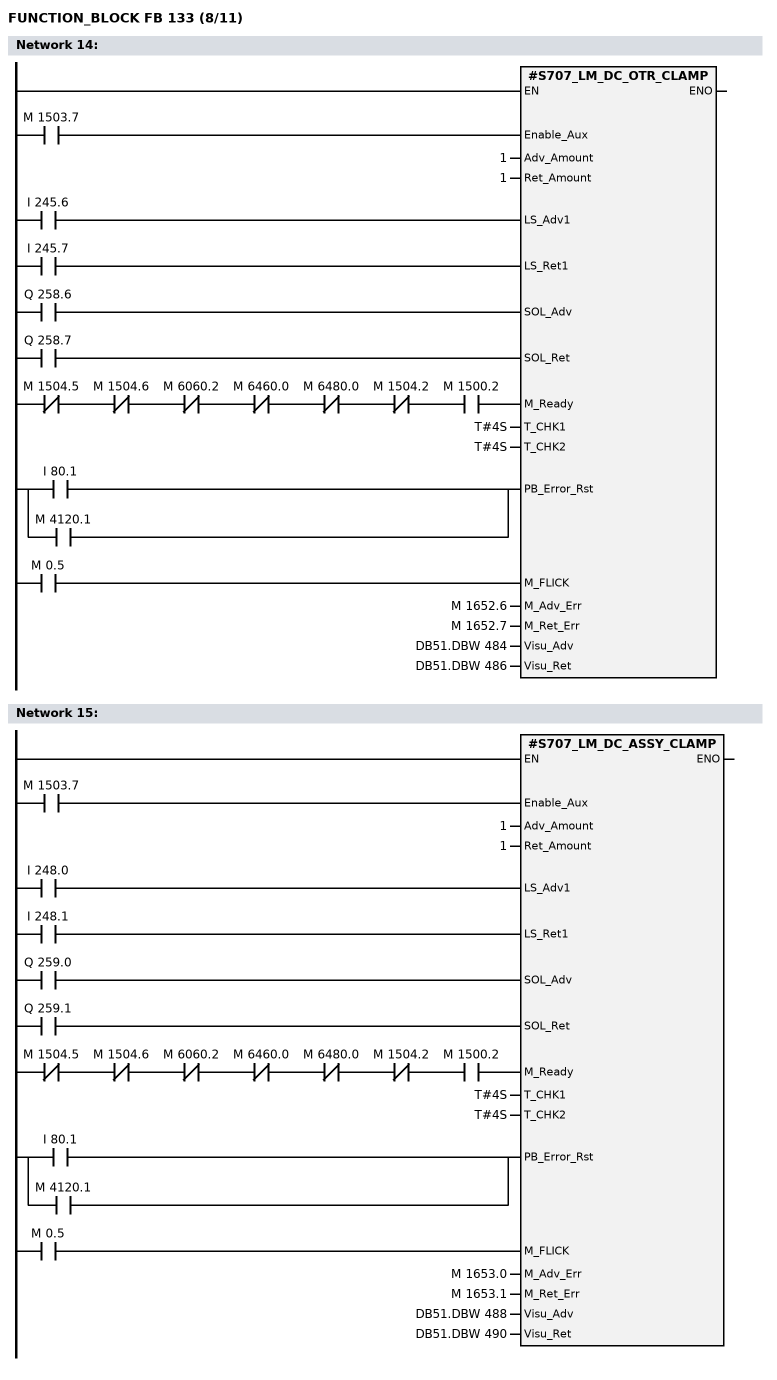

      A     M   1503.7;
      =     L      0.0;
      BLD   103;
      A     I    245.6;
      =     L      0.1;
      BLD   103;
      A     I    245.7;
      =     L      0.2;
      BLD   103;
      A     Q    258.6;
      =     L      1.1;
      BLD   103;
      A     Q    258.7;
      =     L      1.2;
      BLD   103;
      AN    M   1504.5;
      AN    M   1504.6;
      AN    M   6060.2;
      AN    M   6460.0;
      AN    M   6480.0;
      AN    M   1504.2;
      A     M   1500.2;
      =     L      1.3;
      BLD   103;
      A(    ;
      O     I     80.1;
      O     M   4120.1;
      )     ;
      =     L      1.5;
      BLD   103;
      A     M      0.5;
      =     L      1.6;
      BLD   103;
      CALL #S707_LM_DC_OTR_CLAMP (
           Enable_Aux               := L      0.0,
           Adv_Amount               := 1,
           Ret_Amount               := 1,
           LS_Adv1                  := L      0.1,
           LS_Ret1                  := L      0.2,
           SOL_Adv                  := L      1.1,
           SOL_Ret                  := L      1.2,
           M_Ready                  := L      1.3,
           T_CHK1                   := T#4S,
           T_CHK2                   := T#4S,
           PB_Error_Rst             := L      1.5,
           M_FLICK                  := L      1.6,
           M_Adv_Err                := M   1652.6,
           M_Ret_Err                := M   1652.7,
           Visu_Adv                 := DB51.DBW  484,
           Visu_Ret                 := DB51.DBW  486);
      NOP   0;
NETWORK
TITLE =

      A     M   1503.7;
      =     L      0.0;
      BLD   103;
      A     I    248.0;
      =     L      0.1;
      BLD   103;
      A     I    248.1;
      =     L      0.2;
      BLD   103;
      A     Q    259.0;
      =     L      1.1;
      BLD   103;
      A     Q    259.1;
      =     L      1.2;
      BLD   103;
      AN    M   1504.5;
      AN    M   1504.6;
      AN    M   6060.2;
      AN    M   6460.0;
      AN    M   6480.0;
      AN    M   1504.2;
      A     M   1500.2;
      =     L      1.3;
      BLD   103;
      A(    ;
      O     I     80.1;
      O     M   4120.1;
      )     ;
      =     L      1.5;
      BLD   103;
      A     M      0.5;
      =     L      1.6;
      BLD   103;
      CALL #S707_LM_DC_ASSY_CLAMP (
           Enable_Aux               := L      0.0,
           Adv_Amount               := 1,
           Ret_Amount               := 1,
           LS_Adv1                  := L      0.1,
           LS_Ret1                  := L      0.2,
           SOL_Adv                  := L      1.1,
           SOL_Ret                  := L      1.2,
           M_Ready                  := L      1.3,
           T_CHK1                   := T#4S,
           T_CHK2                   := T#4S,
           PB_Error_Rst             := L      1.5,
           M_FLICK                  := L      1.6,
           M_Adv_Err                := M   1653.0,
           M_Ret_Err                := M   1653.1,
           Visu_Adv                 := DB51.DBW  488,
           Visu_Ret                 := DB51.DBW  490);
      NOP   0;
NETWORK
TITLE =
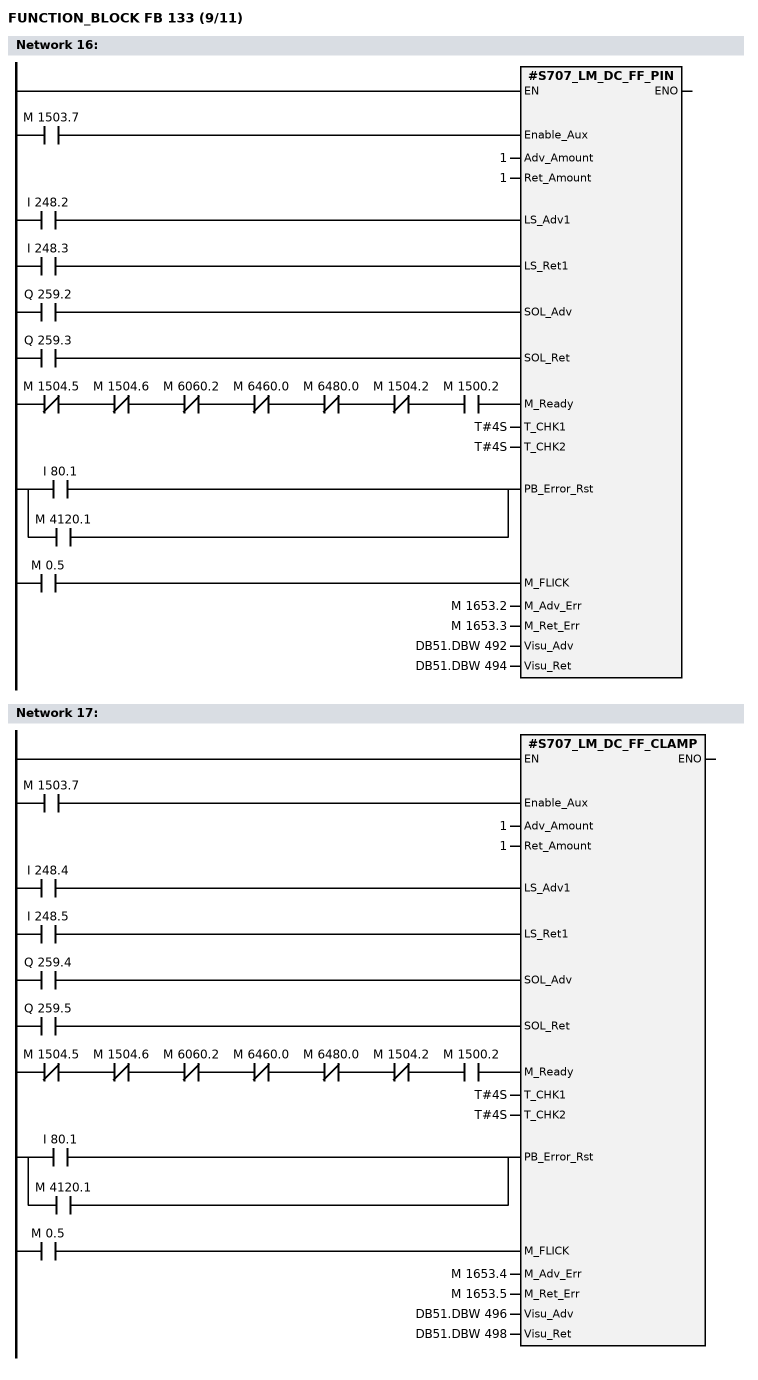

      A     M   1503.7;
      =     L      0.0;
      BLD   103;
      A     I    248.2;
      =     L      0.1;
      BLD   103;
      A     I    248.3;
      =     L      0.2;
      BLD   103;
      A     Q    259.2;
      =     L      1.1;
      BLD   103;
      A     Q    259.3;
      =     L      1.2;
      BLD   103;
      AN    M   1504.5;
      AN    M   1504.6;
      AN    M   6060.2;
      AN    M   6460.0;
      AN    M   6480.0;
      AN    M   1504.2;
      A     M   1500.2;
      =     L      1.3;
      BLD   103;
      A(    ;
      O     I     80.1;
      O     M   4120.1;
      )     ;
      =     L      1.5;
      BLD   103;
      A     M      0.5;
      =     L      1.6;
      BLD   103;
      CALL #S707_LM_DC_FF_PIN (
           Enable_Aux               := L      0.0,
           Adv_Amount               := 1,
           Ret_Amount               := 1,
           LS_Adv1                  := L      0.1,
           LS_Ret1                  := L      0.2,
           SOL_Adv                  := L      1.1,
           SOL_Ret                  := L      1.2,
           M_Ready                  := L      1.3,
           T_CHK1                   := T#4S,
           T_CHK2                   := T#4S,
           PB_Error_Rst             := L      1.5,
           M_FLICK                  := L      1.6,
           M_Adv_Err                := M   1653.2,
           M_Ret_Err                := M   1653.3,
           Visu_Adv                 := DB51.DBW  492,
           Visu_Ret                 := DB51.DBW  494);
      NOP   0;
NETWORK
TITLE =

      A     M   1503.7;
      =     L      0.0;
      BLD   103;
      A     I    248.4;
      =     L      0.1;
      BLD   103;
      A     I    248.5;
      =     L      0.2;
      BLD   103;
      A     Q    259.4;
      =     L      1.1;
      BLD   103;
      A     Q    259.5;
      =     L      1.2;
      BLD   103;
      AN    M   1504.5;
      AN    M   1504.6;
      AN    M   6060.2;
      AN    M   6460.0;
      AN    M   6480.0;
      AN    M   1504.2;
      A     M   1500.2;
      =     L      1.3;
      BLD   103;
      A(    ;
      O     I     80.1;
      O     M   4120.1;
      )     ;
      =     L      1.5;
      BLD   103;
      A     M      0.5;
      =     L      1.6;
      BLD   103;
      CALL #S707_LM_DC_FF_CLAMP (
           Enable_Aux               := L      0.0,
           Adv_Amount               := 1,
           Ret_Amount               := 1,
           LS_Adv1                  := L      0.1,
           LS_Ret1                  := L      0.2,
           SOL_Adv                  := L      1.1,
           SOL_Ret                  := L      1.2,
           M_Ready                  := L      1.3,
           T_CHK1                   := T#4S,
           T_CHK2                   := T#4S,
           PB_Error_Rst             := L      1.5,
           M_FLICK                  := L      1.6,
           M_Adv_Err                := M   1653.4,
           M_Ret_Err                := M   1653.5,
           Visu_Adv                 := DB51.DBW  496,
           Visu_Ret                 := DB51.DBW  498);
      NOP   0;
NETWORK
TITLE =
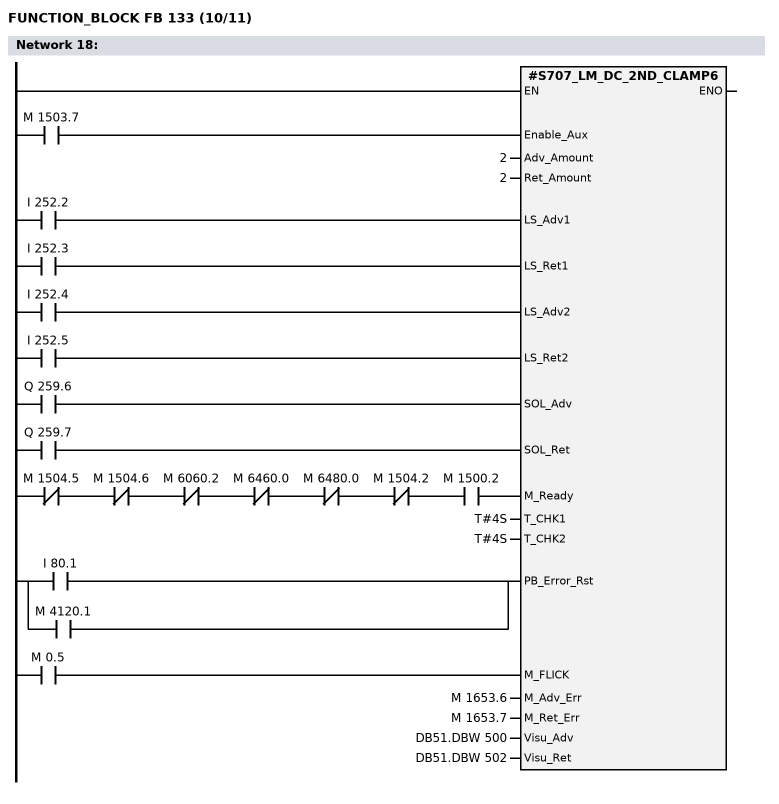

      A     M   1503.7;
      =     L      0.0;
      BLD   103;
      A     I    252.2;
      =     L      0.1;
      BLD   103;
      A     I    252.3;
      =     L      0.2;
      BLD   103;
      A     I    252.4;
      =     L      0.3;
      BLD   103;
      A     I    252.5;
      =     L      0.4;
      BLD   103;
      A     Q    259.6;
      =     L      1.1;
      BLD   103;
      A     Q    259.7;
      =     L      1.2;
      BLD   103;
      AN    M   1504.5;
      AN    M   1504.6;
      AN    M   6060.2;
      AN    M   6460.0;
      AN    M   6480.0;
      AN    M   1504.2;
      A     M   1500.2;
      =     L      1.3;
      BLD   103;
      A(    ;
      O     I     80.1;
      O     M   4120.1;
      )     ;
      =     L      1.5;
      BLD   103;
      A     M      0.5;
      =     L      1.6;
      BLD   103;
      CALL #S707_LM_DC_2ND_CLAMP6 (
           Enable_Aux               := L      0.0,
           Adv_Amount               := 2,
           Ret_Amount               := 2,
           LS_Adv1                  := L      0.1,
           LS_Ret1                  := L      0.2,
           LS_Adv2                  := L      0.3,
           LS_Ret2                  := L      0.4,
           SOL_Adv                  := L      1.1,
           SOL_Ret                  := L      1.2,
           M_Ready                  := L      1.3,
           T_CHK1                   := T#4S,
           T_CHK2                   := T#4S,
           PB_Error_Rst             := L      1.5,
           M_FLICK                  := L      1.6,
           M_Adv_Err                := M   1653.6,
           M_Ret_Err                := M   1653.7,
           Visu_Adv                 := DB51.DBW  500,
           Visu_Ret                 := DB51.DBW  502);
      NOP   0;
NETWORK
TITLE =
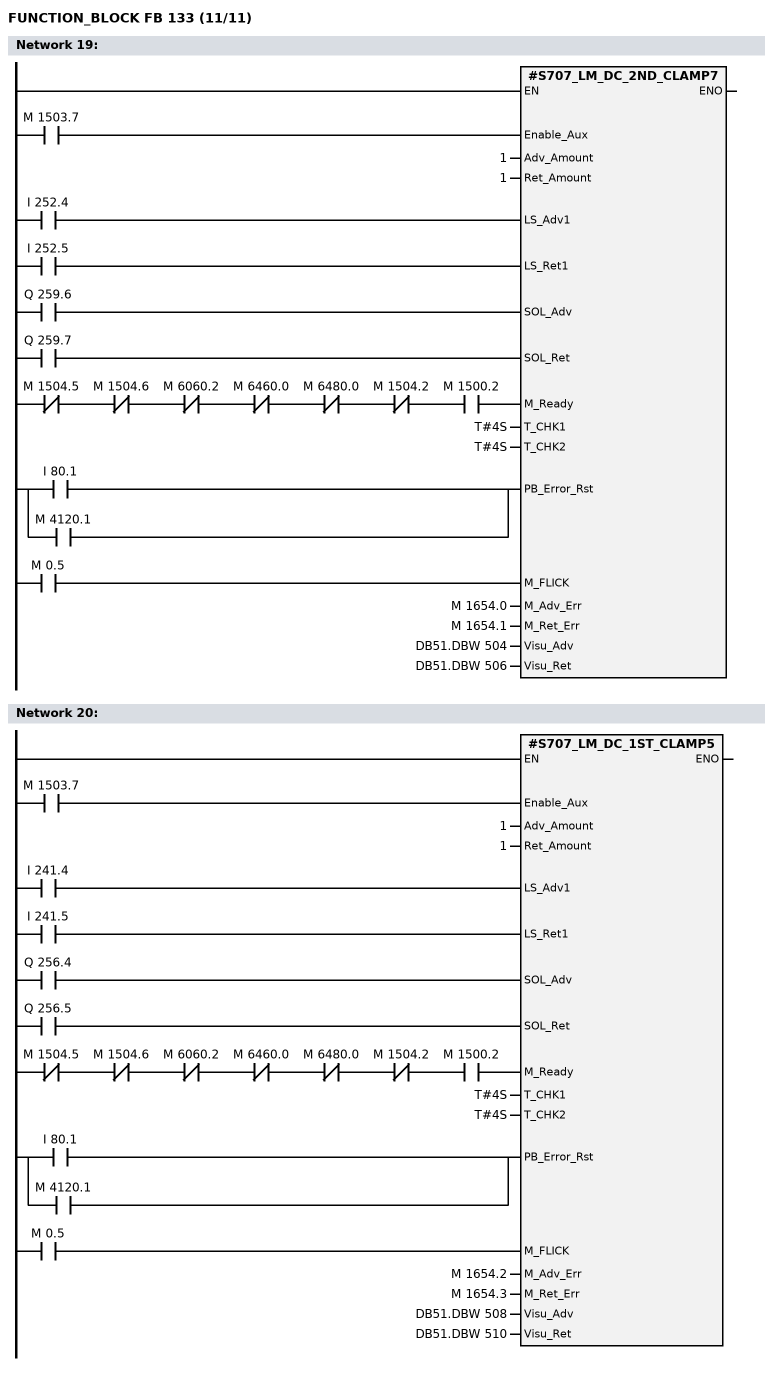

      A     M   1503.7;
      =     L      0.0;
      BLD   103;
      A     I    252.4;
      =     L      0.1;
      BLD   103;
      A     I    252.5;
      =     L      0.2;
      BLD   103;
      A     Q    259.6;
      =     L      1.1;
      BLD   103;
      A     Q    259.7;
      =     L      1.2;
      BLD   103;
      AN    M   1504.5;
      AN    M   1504.6;
      AN    M   6060.2;
      AN    M   6460.0;
      AN    M   6480.0;
      AN    M   1504.2;
      A     M   1500.2;
      =     L      1.3;
      BLD   103;
      A(    ;
      O     I     80.1;
      O     M   4120.1;
      )     ;
      =     L      1.5;
      BLD   103;
      A     M      0.5;
      =     L      1.6;
      BLD   103;
      CALL #S707_LM_DC_2ND_CLAMP7 (
           Enable_Aux               := L      0.0,
           Adv_Amount               := 1,
           Ret_Amount               := 1,
           LS_Adv1                  := L      0.1,
           LS_Ret1                  := L      0.2,
           SOL_Adv                  := L      1.1,
           SOL_Ret                  := L      1.2,
           M_Ready                  := L      1.3,
           T_CHK1                   := T#4S,
           T_CHK2                   := T#4S,
           PB_Error_Rst             := L      1.5,
           M_FLICK                  := L      1.6,
           M_Adv_Err                := M   1654.0,
           M_Ret_Err                := M   1654.1,
           Visu_Adv                 := DB51.DBW  504,
           Visu_Ret                 := DB51.DBW  506);
      NOP   0;
NETWORK
TITLE =

      A     M   1503.7;
      =     L      0.0;
      BLD   103;
      A     I    241.4;
      =     L      0.1;
      BLD   103;
      A     I    241.5;
      =     L      0.2;
      BLD   103;
      A     Q    256.4;
      =     L      1.1;
      BLD   103;
      A     Q    256.5;
      =     L      1.2;
      BLD   103;
      AN    M   1504.5;
      AN    M   1504.6;
      AN    M   6060.2;
      AN    M   6460.0;
      AN    M   6480.0;
      AN    M   1504.2;
      A     M   1500.2;
      =     L      1.3;
      BLD   103;
      A(    ;
      O     I     80.1;
      O     M   4120.1;
      )     ;
      =     L      1.5;
      BLD   103;
      A     M      0.5;
      =     L      1.6;
      BLD   103;
      CALL #S707_LM_DC_1ST_CLAMP5 (
           Enable_Aux               := L      0.0,
           Adv_Amount               := 1,
           Ret_Amount               := 1,
           LS_Adv1                  := L      0.1,
           LS_Ret1                  := L      0.2,
           SOL_Adv                  := L      1.1,
           SOL_Ret                  := L      1.2,
           M_Ready                  := L      1.3,
           T_CHK1                   := T#4S,
           T_CHK2                   := T#4S,
           PB_Error_Rst             := L      1.5,
           M_FLICK                  := L      1.6,
           M_Adv_Err                := M   1654.2,
           M_Ret_Err                := M   1654.3,
           Visu_Adv                 := DB51.DBW  508,
           Visu_Ret                 := DB51.DBW  510);
      NOP   0;
END_FUNCTION_BLOCK

DATA_BLOCK DB 133
TITLE =
VERSION : 0.0

 FB 133
BEGIN
   S707_LM_DC_PIN.Enable_Aux := FALSE;
   S707_LM_DC_PIN.Adv_Amount := 1;
   S707_LM_DC_PIN.Ret_Amount := 1;
   S707_LM_DC_PIN.LS_Adv1 := FALSE;
   S707_LM_DC_PIN.LS_Ret1 := FALSE;
   S707_LM_DC_PIN.LS_Adv2 := FALSE;
   S707_LM_DC_PIN.LS_Ret2 := FALSE;
   S707_LM_DC_PIN.LS_Adv3 := FALSE;
   S707_LM_DC_PIN.LS_Ret3 := FALSE;
   S707_LM_DC_PIN.LS_Adv4 := FALSE;
   S707_LM_DC_PIN.LS_Ret4 := FALSE;
   S707_LM_DC_PIN.SOL_Adv := FALSE;
   S707_LM_DC_PIN.SOL_Ret := FALSE;
   S707_LM_DC_PIN.M_Ready := TRUE;
   S707_LM_DC_PIN.T_CHK1 := T#4S;
   S707_LM_DC_PIN.T_CHK2 := T#4S;
   S707_LM_DC_PIN.PB_Lamp_CHK := FALSE;
   S707_LM_DC_PIN.PB_Error_Rst := FALSE;
   S707_LM_DC_PIN.M_FLICK := TRUE;
   S707_LM_DC_PIN.M_Adv_Err := FALSE;
   S707_LM_DC_PIN.M_Ret_Err := FALSE;
   S707_LM_DC_PIN.LP_Adv := FALSE;
   S707_LM_DC_PIN.LP_Ret := FALSE;
   S707_LM_DC_PIN.Visu_Adv := W#16#0;
   S707_LM_DC_PIN.Visu_Ret := W#16#0;
   S707_LM_DC_PIN.Error_T1.IN := FALSE;
   S707_LM_DC_PIN.Error_T1.PT := T#4S;
   S707_LM_DC_PIN.Error_T1.Q := FALSE;
   S707_LM_DC_PIN.Error_T1.ET := T#0MS;
   S707_LM_DC_PIN.Error_T1.STATE := B#16#0;
   S707_LM_DC_PIN.Error_T1.STIME := T#0MS;
   S707_LM_DC_PIN.Error_T1.ATIME := T#0MS;
   S707_LM_DC_PIN.Error_T2.IN := FALSE;
   S707_LM_DC_PIN.Error_T2.PT := T#4S;
   S707_LM_DC_PIN.Error_T2.Q := FALSE;
   S707_LM_DC_PIN.Error_T2.ET := T#0MS;
   S707_LM_DC_PIN.Error_T2.STATE := B#16#0;
   S707_LM_DC_PIN.Error_T2.STIME := T#0MS;
   S707_LM_DC_PIN.Error_T2.ATIME := T#0MS;
   S707_LM_DC_PIN.CHK_Aux1 := FALSE;
   S707_LM_DC_PIN.CHK_Aux2 := FALSE;
   S707_LM_DC_PIN.Error_T1_DN := FALSE;
   S707_LM_DC_PIN.Error_T2_DN := FALSE;
   S707_LM_DC_PIN.Adv_Memo := TRUE;
   S707_LM_DC_PIN.Visu_Adv_Arr[0] := FALSE;
   S707_LM_DC_PIN.Visu_Adv_Arr[1] := FALSE;
   S707_LM_DC_PIN.Visu_Adv_Arr[2] := FALSE;
   S707_LM_DC_PIN.Visu_Adv_Arr[3] := FALSE;
   S707_LM_DC_PIN.Visu_Adv_Arr[4] := FALSE;
   S707_LM_DC_PIN.Visu_Adv_Arr[5] := FALSE;
   S707_LM_DC_PIN.Visu_Adv_Arr[6] := FALSE;
   S707_LM_DC_PIN.Visu_Adv_Arr[7] := FALSE;
   S707_LM_DC_PIN.Visu_Adv_Arr[8] := FALSE;
   S707_LM_DC_PIN.Visu_Adv_Arr[9] := FALSE;
   S707_LM_DC_PIN.Visu_Adv_Arr[10] := FALSE;
   S707_LM_DC_PIN.Visu_Adv_Arr[11] := FALSE;
   S707_LM_DC_PIN.Visu_Adv_Arr[12] := FALSE;
   S707_LM_DC_PIN.Visu_Adv_Arr[13] := FALSE;
   S707_LM_DC_PIN.Visu_Adv_Arr[14] := FALSE;
   S707_LM_DC_PIN.Visu_Adv_Arr[15] := FALSE;
   S707_LM_DC_PIN.Visu_Ret_Arr[0] := FALSE;
   S707_LM_DC_PIN.Visu_Ret_Arr[1] := FALSE;
   S707_LM_DC_PIN.Visu_Ret_Arr[2] := FALSE;
   S707_LM_DC_PIN.Visu_Ret_Arr[3] := FALSE;
   S707_LM_DC_PIN.Visu_Ret_Arr[4] := FALSE;
   S707_LM_DC_PIN.Visu_Ret_Arr[5] := FALSE;
   S707_LM_DC_PIN.Visu_Ret_Arr[6] := FALSE;
   S707_LM_DC_PIN.Visu_Ret_Arr[7] := FALSE;
   S707_LM_DC_PIN.Visu_Ret_Arr[8] := FALSE;
   S707_LM_DC_PIN.Visu_Ret_Arr[9] := FALSE;
   S707_LM_DC_PIN.Visu_Ret_Arr[10] := FALSE;
   S707_LM_DC_PIN.Visu_Ret_Arr[11] := FALSE;
   S707_LM_DC_PIN.Visu_Ret_Arr[12] := FALSE;
   S707_LM_DC_PIN.Visu_Ret_Arr[13] := FALSE;
   S707_LM_DC_PIN.Visu_Ret_Arr[14] := FALSE;
   S707_LM_DC_PIN.Visu_Ret_Arr[15] := FALSE;
   S707_LM_DC_PIN.BLK_Move_Ret := 0;
   S707_LM_DC_PIN.Enable := FALSE;
   S707_LM_DC_PIN.Adv_End := FALSE;
   S707_LM_DC_PIN.Ret_End := FALSE;
   S707_LM_DC_1ST_CLAMP1.Enable_Aux := FALSE;
   S707_LM_DC_1ST_CLAMP1.Adv_Amount := 1;
   S707_LM_DC_1ST_CLAMP1.Ret_Amount := 1;
   S707_LM_DC_1ST_CLAMP1.LS_Adv1 := FALSE;
   S707_LM_DC_1ST_CLAMP1.LS_Ret1 := FALSE;
   S707_LM_DC_1ST_CLAMP1.LS_Adv2 := FALSE;
   S707_LM_DC_1ST_CLAMP1.LS_Ret2 := FALSE;
   S707_LM_DC_1ST_CLAMP1.LS_Adv3 := FALSE;
   S707_LM_DC_1ST_CLAMP1.LS_Ret3 := FALSE;
   S707_LM_DC_1ST_CLAMP1.LS_Adv4 := FALSE;
   S707_LM_DC_1ST_CLAMP1.LS_Ret4 := FALSE;
   S707_LM_DC_1ST_CLAMP1.SOL_Adv := FALSE;
   S707_LM_DC_1ST_CLAMP1.SOL_Ret := FALSE;
   S707_LM_DC_1ST_CLAMP1.M_Ready := TRUE;
   S707_LM_DC_1ST_CLAMP1.T_CHK1 := T#4S;
   S707_LM_DC_1ST_CLAMP1.T_CHK2 := T#4S;
   S707_LM_DC_1ST_CLAMP1.PB_Lamp_CHK := FALSE;
   S707_LM_DC_1ST_CLAMP1.PB_Error_Rst := FALSE;
   S707_LM_DC_1ST_CLAMP1.M_FLICK := TRUE;
   S707_LM_DC_1ST_CLAMP1.M_Adv_Err := FALSE;
   S707_LM_DC_1ST_CLAMP1.M_Ret_Err := FALSE;
   S707_LM_DC_1ST_CLAMP1.LP_Adv := FALSE;
   S707_LM_DC_1ST_CLAMP1.LP_Ret := FALSE;
   S707_LM_DC_1ST_CLAMP1.Visu_Adv := W#16#0;
   S707_LM_DC_1ST_CLAMP1.Visu_Ret := W#16#0;
   S707_LM_DC_1ST_CLAMP1.Error_T1.IN := FALSE;
   S707_LM_DC_1ST_CLAMP1.Error_T1.PT := T#4S;
   S707_LM_DC_1ST_CLAMP1.Error_T1.Q := FALSE;
   S707_LM_DC_1ST_CLAMP1.Error_T1.ET := T#0MS;
   S707_LM_DC_1ST_CLAMP1.Error_T1.STATE := B#16#0;
   S707_LM_DC_1ST_CLAMP1.Error_T1.STIME := T#0MS;
   S707_LM_DC_1ST_CLAMP1.Error_T1.ATIME := T#0MS;
   S707_LM_DC_1ST_CLAMP1.Error_T2.IN := FALSE;
   S707_LM_DC_1ST_CLAMP1.Error_T2.PT := T#4S;
   S707_LM_DC_1ST_CLAMP1.Error_T2.Q := FALSE;
   S707_LM_DC_1ST_CLAMP1.Error_T2.ET := T#0MS;
   S707_LM_DC_1ST_CLAMP1.Error_T2.STATE := B#16#0;
   S707_LM_DC_1ST_CLAMP1.Error_T2.STIME := T#0MS;
   S707_LM_DC_1ST_CLAMP1.Error_T2.ATIME := T#0MS;
   S707_LM_DC_1ST_CLAMP1.CHK_Aux1 := FALSE;
   S707_LM_DC_1ST_CLAMP1.CHK_Aux2 := FALSE;
   S707_LM_DC_1ST_CLAMP1.Error_T1_DN := FALSE;
   S707_LM_DC_1ST_CLAMP1.Error_T2_DN := FALSE;
   S707_LM_DC_1ST_CLAMP1.Adv_Memo := TRUE;
   S707_LM_DC_1ST_CLAMP1.Visu_Adv_Arr[0] := FALSE;
   S707_LM_DC_1ST_CLAMP1.Visu_Adv_Arr[1] := FALSE;
   S707_LM_DC_1ST_CLAMP1.Visu_Adv_Arr[2] := FALSE;
   S707_LM_DC_1ST_CLAMP1.Visu_Adv_Arr[3] := FALSE;
   S707_LM_DC_1ST_CLAMP1.Visu_Adv_Arr[4] := FALSE;
   S707_LM_DC_1ST_CLAMP1.Visu_Adv_Arr[5] := FALSE;
   S707_LM_DC_1ST_CLAMP1.Visu_Adv_Arr[6] := FALSE;
   S707_LM_DC_1ST_CLAMP1.Visu_Adv_Arr[7] := FALSE;
   S707_LM_DC_1ST_CLAMP1.Visu_Adv_Arr[8] := FALSE;
   S707_LM_DC_1ST_CLAMP1.Visu_Adv_Arr[9] := FALSE;
   S707_LM_DC_1ST_CLAMP1.Visu_Adv_Arr[10] := FALSE;
   S707_LM_DC_1ST_CLAMP1.Visu_Adv_Arr[11] := FALSE;
   S707_LM_DC_1ST_CLAMP1.Visu_Adv_Arr[12] := FALSE;
   S707_LM_DC_1ST_CLAMP1.Visu_Adv_Arr[13] := FALSE;
   S707_LM_DC_1ST_CLAMP1.Visu_Adv_Arr[14] := FALSE;
   S707_LM_DC_1ST_CLAMP1.Visu_Adv_Arr[15] := FALSE;
   S707_LM_DC_1ST_CLAMP1.Visu_Ret_Arr[0] := FALSE;
   S707_LM_DC_1ST_CLAMP1.Visu_Ret_Arr[1] := FALSE;
   S707_LM_DC_1ST_CLAMP1.Visu_Ret_Arr[2] := FALSE;
   S707_LM_DC_1ST_CLAMP1.Visu_Ret_Arr[3] := FALSE;
   S707_LM_DC_1ST_CLAMP1.Visu_Ret_Arr[4] := FALSE;
   S707_LM_DC_1ST_CLAMP1.Visu_Ret_Arr[5] := FALSE;
   S707_LM_DC_1ST_CLAMP1.Visu_Ret_Arr[6] := FALSE;
   S707_LM_DC_1ST_CLAMP1.Visu_Ret_Arr[7] := FALSE;
   S707_LM_DC_1ST_CLAMP1.Visu_Ret_Arr[8] := FALSE;
   S707_LM_DC_1ST_CLAMP1.Visu_Ret_Arr[9] := FALSE;
   S707_LM_DC_1ST_CLAMP1.Visu_Ret_Arr[10] := FALSE;
   S707_LM_DC_1ST_CLAMP1.Visu_Ret_Arr[11] := FALSE;
   S707_LM_DC_1ST_CLAMP1.Visu_Ret_Arr[12] := FALSE;
   S707_LM_DC_1ST_CLAMP1.Visu_Ret_Arr[13] := FALSE;
   S707_LM_DC_1ST_CLAMP1.Visu_Ret_Arr[14] := FALSE;
   S707_LM_DC_1ST_CLAMP1.Visu_Ret_Arr[15] := FALSE;
   S707_LM_DC_1ST_CLAMP1.BLK_Move_Ret := 0;
   S707_LM_DC_1ST_CLAMP1.Enable := FALSE;
   S707_LM_DC_1ST_CLAMP1.Adv_End := FALSE;
   S707_LM_DC_1ST_CLAMP1.Ret_End := FALSE;
   S707_LM_DC_1ST_CLAMP2.Enable_Aux := FALSE;
   S707_LM_DC_1ST_CLAMP2.Adv_Amount := 2;
   S707_LM_DC_1ST_CLAMP2.Ret_Amount := 2;
   S707_LM_DC_1ST_CLAMP2.LS_Adv1 := FALSE;
   S707_LM_DC_1ST_CLAMP2.LS_Ret1 := FALSE;
   S707_LM_DC_1ST_CLAMP2.LS_Adv2 := FALSE;
   S707_LM_DC_1ST_CLAMP2.LS_Ret2 := FALSE;
   S707_LM_DC_1ST_CLAMP2.LS_Adv3 := FALSE;
   S707_LM_DC_1ST_CLAMP2.LS_Ret3 := FALSE;
   S707_LM_DC_1ST_CLAMP2.LS_Adv4 := FALSE;
   S707_LM_DC_1ST_CLAMP2.LS_Ret4 := FALSE;
   S707_LM_DC_1ST_CLAMP2.SOL_Adv := FALSE;
   S707_LM_DC_1ST_CLAMP2.SOL_Ret := FALSE;
   S707_LM_DC_1ST_CLAMP2.M_Ready := TRUE;
   S707_LM_DC_1ST_CLAMP2.T_CHK1 := T#4S;
   S707_LM_DC_1ST_CLAMP2.T_CHK2 := T#4S;
   S707_LM_DC_1ST_CLAMP2.PB_Lamp_CHK := FALSE;
   S707_LM_DC_1ST_CLAMP2.PB_Error_Rst := FALSE;
   S707_LM_DC_1ST_CLAMP2.M_FLICK := TRUE;
   S707_LM_DC_1ST_CLAMP2.M_Adv_Err := FALSE;
   S707_LM_DC_1ST_CLAMP2.M_Ret_Err := FALSE;
   S707_LM_DC_1ST_CLAMP2.LP_Adv := FALSE;
   S707_LM_DC_1ST_CLAMP2.LP_Ret := FALSE;
   S707_LM_DC_1ST_CLAMP2.Visu_Adv := W#16#0;
   S707_LM_DC_1ST_CLAMP2.Visu_Ret := W#16#0;
   S707_LM_DC_1ST_CLAMP2.Error_T1.IN := FALSE;
   S707_LM_DC_1ST_CLAMP2.Error_T1.PT := T#4S;
   S707_LM_DC_1ST_CLAMP2.Error_T1.Q := FALSE;
   S707_LM_DC_1ST_CLAMP2.Error_T1.ET := T#0MS;
   S707_LM_DC_1ST_CLAMP2.Error_T1.STATE := B#16#0;
   S707_LM_DC_1ST_CLAMP2.Error_T1.STIME := T#0MS;
   S707_LM_DC_1ST_CLAMP2.Error_T1.ATIME := T#0MS;
   S707_LM_DC_1ST_CLAMP2.Error_T2.IN := FALSE;
   S707_LM_DC_1ST_CLAMP2.Error_T2.PT := T#4S;
   S707_LM_DC_1ST_CLAMP2.Error_T2.Q := FALSE;
   S707_LM_DC_1ST_CLAMP2.Error_T2.ET := T#0MS;
   S707_LM_DC_1ST_CLAMP2.Error_T2.STATE := B#16#0;
   S707_LM_DC_1ST_CLAMP2.Error_T2.STIME := T#0MS;
   S707_LM_DC_1ST_CLAMP2.Error_T2.ATIME := T#0MS;
   S707_LM_DC_1ST_CLAMP2.CHK_Aux1 := FALSE;
   S707_LM_DC_1ST_CLAMP2.CHK_Aux2 := FALSE;
   S707_LM_DC_1ST_CLAMP2.Error_T1_DN := FALSE;
   S707_LM_DC_1ST_CLAMP2.Error_T2_DN := FALSE;
   S707_LM_DC_1ST_CLAMP2.Adv_Memo := TRUE;
   S707_LM_DC_1ST_CLAMP2.Visu_Adv_Arr[0] := FALSE;
   S707_LM_DC_1ST_CLAMP2.Visu_Adv_Arr[1] := FALSE;
   S707_LM_DC_1ST_CLAMP2.Visu_Adv_Arr[2] := FALSE;
   S707_LM_DC_1ST_CLAMP2.Visu_Adv_Arr[3] := FALSE;
   S707_LM_DC_1ST_CLAMP2.Visu_Adv_Arr[4] := FALSE;
   S707_LM_DC_1ST_CLAMP2.Visu_Adv_Arr[5] := FALSE;
   S707_LM_DC_1ST_CLAMP2.Visu_Adv_Arr[6] := FALSE;
   S707_LM_DC_1ST_CLAMP2.Visu_Adv_Arr[7] := FALSE;
   S707_LM_DC_1ST_CLAMP2.Visu_Adv_Arr[8] := FALSE;
   S707_LM_DC_1ST_CLAMP2.Visu_Adv_Arr[9] := FALSE;
   S707_LM_DC_1ST_CLAMP2.Visu_Adv_Arr[10] := FALSE;
   S707_LM_DC_1ST_CLAMP2.Visu_Adv_Arr[11] := FALSE;
   S707_LM_DC_1ST_CLAMP2.Visu_Adv_Arr[12] := FALSE;
   S707_LM_DC_1ST_CLAMP2.Visu_Adv_Arr[13] := FALSE;
   S707_LM_DC_1ST_CLAMP2.Visu_Adv_Arr[14] := FALSE;
   S707_LM_DC_1ST_CLAMP2.Visu_Adv_Arr[15] := FALSE;
   S707_LM_DC_1ST_CLAMP2.Visu_Ret_Arr[0] := FALSE;
   S707_LM_DC_1ST_CLAMP2.Visu_Ret_Arr[1] := FALSE;
   S707_LM_DC_1ST_CLAMP2.Visu_Ret_Arr[2] := FALSE;
   S707_LM_DC_1ST_CLAMP2.Visu_Ret_Arr[3] := FALSE;
   S707_LM_DC_1ST_CLAMP2.Visu_Ret_Arr[4] := FALSE;
   S707_LM_DC_1ST_CLAMP2.Visu_Ret_Arr[5] := FALSE;
   S707_LM_DC_1ST_CLAMP2.Visu_Ret_Arr[6] := FALSE;
   S707_LM_DC_1ST_CLAMP2.Visu_Ret_Arr[7] := FALSE;
   S707_LM_DC_1ST_CLAMP2.Visu_Ret_Arr[8] := FALSE;
   S707_LM_DC_1ST_CLAMP2.Visu_Ret_Arr[9] := FALSE;
   S707_LM_DC_1ST_CLAMP2.Visu_Ret_Arr[10] := FALSE;
   S707_LM_DC_1ST_CLAMP2.Visu_Ret_Arr[11] := FALSE;
   S707_LM_DC_1ST_CLAMP2.Visu_Ret_Arr[12] := FALSE;
   S707_LM_DC_1ST_CLAMP2.Visu_Ret_Arr[13] := FALSE;
   S707_LM_DC_1ST_CLAMP2.Visu_Ret_Arr[14] := FALSE;
   S707_LM_DC_1ST_CLAMP2.Visu_Ret_Arr[15] := FALSE;
   S707_LM_DC_1ST_CLAMP2.BLK_Move_Ret := 0;
   S707_LM_DC_1ST_CLAMP2.Enable := FALSE;
   S707_LM_DC_1ST_CLAMP2.Adv_End := FALSE;
   S707_LM_DC_1ST_CLAMP2.Ret_End := FALSE;
   S707_LM_DC_1ST_CLAMP3.Enable_Aux := FALSE;
   S707_LM_DC_1ST_CLAMP3.Adv_Amount := 1;
   S707_LM_DC_1ST_CLAMP3.Ret_Amount := 1;
   S707_LM_DC_1ST_CLAMP3.LS_Adv1 := FALSE;
   S707_LM_DC_1ST_CLAMP3.LS_Ret1 := FALSE;
   S707_LM_DC_1ST_CLAMP3.LS_Adv2 := FALSE;
   S707_LM_DC_1ST_CLAMP3.LS_Ret2 := FALSE;
   S707_LM_DC_1ST_CLAMP3.LS_Adv3 := FALSE;
   S707_LM_DC_1ST_CLAMP3.LS_Ret3 := FALSE;
   S707_LM_DC_1ST_CLAMP3.LS_Adv4 := FALSE;
   S707_LM_DC_1ST_CLAMP3.LS_Ret4 := FALSE;
   S707_LM_DC_1ST_CLAMP3.SOL_Adv := FALSE;
   S707_LM_DC_1ST_CLAMP3.SOL_Ret := FALSE;
   S707_LM_DC_1ST_CLAMP3.M_Ready := TRUE;
   S707_LM_DC_1ST_CLAMP3.T_CHK1 := T#4S;
   S707_LM_DC_1ST_CLAMP3.T_CHK2 := T#4S;
   S707_LM_DC_1ST_CLAMP3.PB_Lamp_CHK := FALSE;
   S707_LM_DC_1ST_CLAMP3.PB_Error_Rst := FALSE;
   S707_LM_DC_1ST_CLAMP3.M_FLICK := TRUE;
   S707_LM_DC_1ST_CLAMP3.M_Adv_Err := FALSE;
   S707_LM_DC_1ST_CLAMP3.M_Ret_Err := FALSE;
   S707_LM_DC_1ST_CLAMP3.LP_Adv := FALSE;
   S707_LM_DC_1ST_CLAMP3.LP_Ret := FALSE;
   S707_LM_DC_1ST_CLAMP3.Visu_Adv := W#16#0;
   S707_LM_DC_1ST_CLAMP3.Visu_Ret := W#16#0;
   S707_LM_DC_1ST_CLAMP3.Error_T1.IN := FALSE;
   S707_LM_DC_1ST_CLAMP3.Error_T1.PT := T#4S;
   S707_LM_DC_1ST_CLAMP3.Error_T1.Q := FALSE;
   S707_LM_DC_1ST_CLAMP3.Error_T1.ET := T#0MS;
   S707_LM_DC_1ST_CLAMP3.Error_T1.STATE := B#16#0;
   S707_LM_DC_1ST_CLAMP3.Error_T1.STIME := T#0MS;
   S707_LM_DC_1ST_CLAMP3.Error_T1.ATIME := T#0MS;
   S707_LM_DC_1ST_CLAMP3.Error_T2.IN := FALSE;
   S707_LM_DC_1ST_CLAMP3.Error_T2.PT := T#4S;
   S707_LM_DC_1ST_CLAMP3.Error_T2.Q := FALSE;
   S707_LM_DC_1ST_CLAMP3.Error_T2.ET := T#0MS;
   S707_LM_DC_1ST_CLAMP3.Error_T2.STATE := B#16#0;
   S707_LM_DC_1ST_CLAMP3.Error_T2.STIME := T#0MS;
   S707_LM_DC_1ST_CLAMP3.Error_T2.ATIME := T#0MS;
   S707_LM_DC_1ST_CLAMP3.CHK_Aux1 := FALSE;
   S707_LM_DC_1ST_CLAMP3.CHK_Aux2 := FALSE;
   S707_LM_DC_1ST_CLAMP3.Error_T1_DN := FALSE;
   S707_LM_DC_1ST_CLAMP3.Error_T2_DN := FALSE;
   S707_LM_DC_1ST_CLAMP3.Adv_Memo := FALSE;
   S707_LM_DC_1ST_CLAMP3.Visu_Adv_Arr[0] := FALSE;
   S707_LM_DC_1ST_CLAMP3.Visu_Adv_Arr[1] := FALSE;
   S707_LM_DC_1ST_CLAMP3.Visu_Adv_Arr[2] := FALSE;
   S707_LM_DC_1ST_CLAMP3.Visu_Adv_Arr[3] := FALSE;
   S707_LM_DC_1ST_CLAMP3.Visu_Adv_Arr[4] := FALSE;
   S707_LM_DC_1ST_CLAMP3.Visu_Adv_Arr[5] := FALSE;
   S707_LM_DC_1ST_CLAMP3.Visu_Adv_Arr[6] := FALSE;
   S707_LM_DC_1ST_CLAMP3.Visu_Adv_Arr[7] := FALSE;
   S707_LM_DC_1ST_CLAMP3.Visu_Adv_Arr[8] := FALSE;
   S707_LM_DC_1ST_CLAMP3.Visu_Adv_Arr[9] := FALSE;
   S707_LM_DC_1ST_CLAMP3.Visu_Adv_Arr[10] := FALSE;
   S707_LM_DC_1ST_CLAMP3.Visu_Adv_Arr[11] := FALSE;
   S707_LM_DC_1ST_CLAMP3.Visu_Adv_Arr[12] := FALSE;
   S707_LM_DC_1ST_CLAMP3.Visu_Adv_Arr[13] := FALSE;
   S707_LM_DC_1ST_CLAMP3.Visu_Adv_Arr[14] := FALSE;
   S707_LM_DC_1ST_CLAMP3.Visu_Adv_Arr[15] := FALSE;
   S707_LM_DC_1ST_CLAMP3.Visu_Ret_Arr[0] := FALSE;
   S707_LM_DC_1ST_CLAMP3.Visu_Ret_Arr[1] := FALSE;
   S707_LM_DC_1ST_CLAMP3.Visu_Ret_Arr[2] := FALSE;
   S707_LM_DC_1ST_CLAMP3.Visu_Ret_Arr[3] := FALSE;
   S707_LM_DC_1ST_CLAMP3.Visu_Ret_Arr[4] := FALSE;
   S707_LM_DC_1ST_CLAMP3.Visu_Ret_Arr[5] := FALSE;
   S707_LM_DC_1ST_CLAMP3.Visu_Ret_Arr[6] := FALSE;
   S707_LM_DC_1ST_CLAMP3.Visu_Ret_Arr[7] := FALSE;
   S707_LM_DC_1ST_CLAMP3.Visu_Ret_Arr[8] := FALSE;
   S707_LM_DC_1ST_CLAMP3.Visu_Ret_Arr[9] := FALSE;
   S707_LM_DC_1ST_CLAMP3.Visu_Ret_Arr[10] := FALSE;
   S707_LM_DC_1ST_CLAMP3.Visu_Ret_Arr[11] := FALSE;
   S707_LM_DC_1ST_CLAMP3.Visu_Ret_Arr[12] := FALSE;
   S707_LM_DC_1ST_CLAMP3.Visu_Ret_Arr[13] := FALSE;
   S707_LM_DC_1ST_CLAMP3.Visu_Ret_Arr[14] := FALSE;
   S707_LM_DC_1ST_CLAMP3.Visu_Ret_Arr[15] := FALSE;
   S707_LM_DC_1ST_CLAMP3.BLK_Move_Ret := 0;
   S707_LM_DC_1ST_CLAMP3.Enable := FALSE;
   S707_LM_DC_1ST_CLAMP3.Adv_End := FALSE;
   S707_LM_DC_1ST_CLAMP3.Ret_End := FALSE;
   S707_LM_DC_1ST_CLAMP4.Enable_Aux := FALSE;
   S707_LM_DC_1ST_CLAMP4.Adv_Amount := 1;
   S707_LM_DC_1ST_CLAMP4.Ret_Amount := 1;
   S707_LM_DC_1ST_CLAMP4.LS_Adv1 := FALSE;
   S707_LM_DC_1ST_CLAMP4.LS_Ret1 := FALSE;
   S707_LM_DC_1ST_CLAMP4.LS_Adv2 := FALSE;
   S707_LM_DC_1ST_CLAMP4.LS_Ret2 := FALSE;
   S707_LM_DC_1ST_CLAMP4.LS_Adv3 := FALSE;
   S707_LM_DC_1ST_CLAMP4.LS_Ret3 := FALSE;
   S707_LM_DC_1ST_CLAMP4.LS_Adv4 := FALSE;
   S707_LM_DC_1ST_CLAMP4.LS_Ret4 := FALSE;
   S707_LM_DC_1ST_CLAMP4.SOL_Adv := FALSE;
   S707_LM_DC_1ST_CLAMP4.SOL_Ret := FALSE;
   S707_LM_DC_1ST_CLAMP4.M_Ready := TRUE;
   S707_LM_DC_1ST_CLAMP4.T_CHK1 := T#4S;
   S707_LM_DC_1ST_CLAMP4.T_CHK2 := T#4S;
   S707_LM_DC_1ST_CLAMP4.PB_Lamp_CHK := FALSE;
   S707_LM_DC_1ST_CLAMP4.PB_Error_Rst := FALSE;
   S707_LM_DC_1ST_CLAMP4.M_FLICK := TRUE;
   S707_LM_DC_1ST_CLAMP4.M_Adv_Err := FALSE;
   S707_LM_DC_1ST_CLAMP4.M_Ret_Err := FALSE;
   S707_LM_DC_1ST_CLAMP4.LP_Adv := FALSE;
   S707_LM_DC_1ST_CLAMP4.LP_Ret := FALSE;
   S707_LM_DC_1ST_CLAMP4.Visu_Adv := W#16#0;
   S707_LM_DC_1ST_CLAMP4.Visu_Ret := W#16#0;
   S707_LM_DC_1ST_CLAMP4.Error_T1.IN := FALSE;
   S707_LM_DC_1ST_CLAMP4.Error_T1.PT := T#4S;
   S707_LM_DC_1ST_CLAMP4.Error_T1.Q := FALSE;
   S707_LM_DC_1ST_CLAMP4.Error_T1.ET := T#0MS;
   S707_LM_DC_1ST_CLAMP4.Error_T1.STATE := B#16#0;
   S707_LM_DC_1ST_CLAMP4.Error_T1.STIME := T#0MS;
   S707_LM_DC_1ST_CLAMP4.Error_T1.ATIME := T#0MS;
   S707_LM_DC_1ST_CLAMP4.Error_T2.IN := FALSE;
   S707_LM_DC_1ST_CLAMP4.Error_T2.PT := T#4S;
   S707_LM_DC_1ST_CLAMP4.Error_T2.Q := FALSE;
   S707_LM_DC_1ST_CLAMP4.Error_T2.ET := T#0MS;
   S707_LM_DC_1ST_CLAMP4.Error_T2.STATE := B#16#0;
   S707_LM_DC_1ST_CLAMP4.Error_T2.STIME := T#0MS;
   S707_LM_DC_1ST_CLAMP4.Error_T2.ATIME := T#0MS;
   S707_LM_DC_1ST_CLAMP4.CHK_Aux1 := FALSE;
   S707_LM_DC_1ST_CLAMP4.CHK_Aux2 := FALSE;
   S707_LM_DC_1ST_CLAMP4.Error_T1_DN := FALSE;
   S707_LM_DC_1ST_CLAMP4.Error_T2_DN := FALSE;
   S707_LM_DC_1ST_CLAMP4.Adv_Memo := FALSE;
   S707_LM_DC_1ST_CLAMP4.Visu_Adv_Arr[0] := FALSE;
   S707_LM_DC_1ST_CLAMP4.Visu_Adv_Arr[1] := FALSE;
   S707_LM_DC_1ST_CLAMP4.Visu_Adv_Arr[2] := FALSE;
   S707_LM_DC_1ST_CLAMP4.Visu_Adv_Arr[3] := FALSE;
   S707_LM_DC_1ST_CLAMP4.Visu_Adv_Arr[4] := FALSE;
   S707_LM_DC_1ST_CLAMP4.Visu_Adv_Arr[5] := FALSE;
   S707_LM_DC_1ST_CLAMP4.Visu_Adv_Arr[6] := FALSE;
   S707_LM_DC_1ST_CLAMP4.Visu_Adv_Arr[7] := FALSE;
   S707_LM_DC_1ST_CLAMP4.Visu_Adv_Arr[8] := FALSE;
   S707_LM_DC_1ST_CLAMP4.Visu_Adv_Arr[9] := FALSE;
   S707_LM_DC_1ST_CLAMP4.Visu_Adv_Arr[10] := FALSE;
   S707_LM_DC_1ST_CLAMP4.Visu_Adv_Arr[11] := FALSE;
   S707_LM_DC_1ST_CLAMP4.Visu_Adv_Arr[12] := FALSE;
   S707_LM_DC_1ST_CLAMP4.Visu_Adv_Arr[13] := FALSE;
   S707_LM_DC_1ST_CLAMP4.Visu_Adv_Arr[14] := FALSE;
   S707_LM_DC_1ST_CLAMP4.Visu_Adv_Arr[15] := FALSE;
   S707_LM_DC_1ST_CLAMP4.Visu_Ret_Arr[0] := FALSE;
   S707_LM_DC_1ST_CLAMP4.Visu_Ret_Arr[1] := FALSE;
   S707_LM_DC_1ST_CLAMP4.Visu_Ret_Arr[2] := FALSE;
   S707_LM_DC_1ST_CLAMP4.Visu_Ret_Arr[3] := FALSE;
   S707_LM_DC_1ST_CLAMP4.Visu_Ret_Arr[4] := FALSE;
   S707_LM_DC_1ST_CLAMP4.Visu_Ret_Arr[5] := FALSE;
   S707_LM_DC_1ST_CLAMP4.Visu_Ret_Arr[6] := FALSE;
   S707_LM_DC_1ST_CLAMP4.Visu_Ret_Arr[7] := FALSE;
   S707_LM_DC_1ST_CLAMP4.Visu_Ret_Arr[8] := FALSE;
   S707_LM_DC_1ST_CLAMP4.Visu_Ret_Arr[9] := FALSE;
   S707_LM_DC_1ST_CLAMP4.Visu_Ret_Arr[10] := FALSE;
   S707_LM_DC_1ST_CLAMP4.Visu_Ret_Arr[11] := FALSE;
   S707_LM_DC_1ST_CLAMP4.Visu_Ret_Arr[12] := FALSE;
   S707_LM_DC_1ST_CLAMP4.Visu_Ret_Arr[13] := FALSE;
   S707_LM_DC_1ST_CLAMP4.Visu_Ret_Arr[14] := FALSE;
   S707_LM_DC_1ST_CLAMP4.Visu_Ret_Arr[15] := FALSE;
   S707_LM_DC_1ST_CLAMP4.BLK_Move_Ret := 0;
   S707_LM_DC_1ST_CLAMP4.Enable := FALSE;
   S707_LM_DC_1ST_CLAMP4.Adv_End := FALSE;
   S707_LM_DC_1ST_CLAMP4.Ret_End := FALSE;
   S707_LM_DC_2ND_CLAMP1.Enable_Aux := FALSE;
   S707_LM_DC_2ND_CLAMP1.Adv_Amount := 1;
   S707_LM_DC_2ND_CLAMP1.Ret_Amount := 1;
   S707_LM_DC_2ND_CLAMP1.LS_Adv1 := FALSE;
   S707_LM_DC_2ND_CLAMP1.LS_Ret1 := FALSE;
   S707_LM_DC_2ND_CLAMP1.LS_Adv2 := FALSE;
   S707_LM_DC_2ND_CLAMP1.LS_Ret2 := FALSE;
   S707_LM_DC_2ND_CLAMP1.LS_Adv3 := FALSE;
   S707_LM_DC_2ND_CLAMP1.LS_Ret3 := FALSE;
   S707_LM_DC_2ND_CLAMP1.LS_Adv4 := FALSE;
   S707_LM_DC_2ND_CLAMP1.LS_Ret4 := FALSE;
   S707_LM_DC_2ND_CLAMP1.SOL_Adv := FALSE;
   S707_LM_DC_2ND_CLAMP1.SOL_Ret := FALSE;
   S707_LM_DC_2ND_CLAMP1.M_Ready := TRUE;
   S707_LM_DC_2ND_CLAMP1.T_CHK1 := T#4S;
   S707_LM_DC_2ND_CLAMP1.T_CHK2 := T#4S;
   S707_LM_DC_2ND_CLAMP1.PB_Lamp_CHK := FALSE;
   S707_LM_DC_2ND_CLAMP1.PB_Error_Rst := FALSE;
   S707_LM_DC_2ND_CLAMP1.M_FLICK := TRUE;
   S707_LM_DC_2ND_CLAMP1.M_Adv_Err := FALSE;
   S707_LM_DC_2ND_CLAMP1.M_Ret_Err := FALSE;
   S707_LM_DC_2ND_CLAMP1.LP_Adv := FALSE;
   S707_LM_DC_2ND_CLAMP1.LP_Ret := FALSE;
   S707_LM_DC_2ND_CLAMP1.Visu_Adv := W#16#0;
   S707_LM_DC_2ND_CLAMP1.Visu_Ret := W#16#0;
   S707_LM_DC_2ND_CLAMP1.Error_T1.IN := FALSE;
   S707_LM_DC_2ND_CLAMP1.Error_T1.PT := T#4S;
   S707_LM_DC_2ND_CLAMP1.Error_T1.Q := FALSE;
   S707_LM_DC_2ND_CLAMP1.Error_T1.ET := T#0MS;
   S707_LM_DC_2ND_CLAMP1.Error_T1.STATE := B#16#0;
   S707_LM_DC_2ND_CLAMP1.Error_T1.STIME := T#0MS;
   S707_LM_DC_2ND_CLAMP1.Error_T1.ATIME := T#0MS;
   S707_LM_DC_2ND_CLAMP1.Error_T2.IN := FALSE;
   S707_LM_DC_2ND_CLAMP1.Error_T2.PT := T#4S;
   S707_LM_DC_2ND_CLAMP1.Error_T2.Q := FALSE;
   S707_LM_DC_2ND_CLAMP1.Error_T2.ET := T#0MS;
   S707_LM_DC_2ND_CLAMP1.Error_T2.STATE := B#16#0;
   S707_LM_DC_2ND_CLAMP1.Error_T2.STIME := T#0MS;
   S707_LM_DC_2ND_CLAMP1.Error_T2.ATIME := T#0MS;
   S707_LM_DC_2ND_CLAMP1.CHK_Aux1 := FALSE;
   S707_LM_DC_2ND_CLAMP1.CHK_Aux2 := FALSE;
   S707_LM_DC_2ND_CLAMP1.Error_T1_DN := FALSE;
   S707_LM_DC_2ND_CLAMP1.Error_T2_DN := FALSE;
   S707_LM_DC_2ND_CLAMP1.Adv_Memo := TRUE;
   S707_LM_DC_2ND_CLAMP1.Visu_Adv_Arr[0] := FALSE;
   S707_LM_DC_2ND_CLAMP1.Visu_Adv_Arr[1] := FALSE;
   S707_LM_DC_2ND_CLAMP1.Visu_Adv_Arr[2] := FALSE;
   S707_LM_DC_2ND_CLAMP1.Visu_Adv_Arr[3] := FALSE;
   S707_LM_DC_2ND_CLAMP1.Visu_Adv_Arr[4] := FALSE;
   S707_LM_DC_2ND_CLAMP1.Visu_Adv_Arr[5] := FALSE;
   S707_LM_DC_2ND_CLAMP1.Visu_Adv_Arr[6] := FALSE;
   S707_LM_DC_2ND_CLAMP1.Visu_Adv_Arr[7] := FALSE;
   S707_LM_DC_2ND_CLAMP1.Visu_Adv_Arr[8] := FALSE;
   S707_LM_DC_2ND_CLAMP1.Visu_Adv_Arr[9] := FALSE;
   S707_LM_DC_2ND_CLAMP1.Visu_Adv_Arr[10] := FALSE;
   S707_LM_DC_2ND_CLAMP1.Visu_Adv_Arr[11] := FALSE;
   S707_LM_DC_2ND_CLAMP1.Visu_Adv_Arr[12] := FALSE;
   S707_LM_DC_2ND_CLAMP1.Visu_Adv_Arr[13] := FALSE;
   S707_LM_DC_2ND_CLAMP1.Visu_Adv_Arr[14] := FALSE;
   S707_LM_DC_2ND_CLAMP1.Visu_Adv_Arr[15] := FALSE;
   S707_LM_DC_2ND_CLAMP1.Visu_Ret_Arr[0] := FALSE;
   S707_LM_DC_2ND_CLAMP1.Visu_Ret_Arr[1] := FALSE;
   S707_LM_DC_2ND_CLAMP1.Visu_Ret_Arr[2] := FALSE;
   S707_LM_DC_2ND_CLAMP1.Visu_Ret_Arr[3] := FALSE;
   S707_LM_DC_2ND_CLAMP1.Visu_Ret_Arr[4] := FALSE;
   S707_LM_DC_2ND_CLAMP1.Visu_Ret_Arr[5] := FALSE;
   S707_LM_DC_2ND_CLAMP1.Visu_Ret_Arr[6] := FALSE;
   S707_LM_DC_2ND_CLAMP1.Visu_Ret_Arr[7] := FALSE;
   S707_LM_DC_2ND_CLAMP1.Visu_Ret_Arr[8] := FALSE;
   S707_LM_DC_2ND_CLAMP1.Visu_Ret_Arr[9] := FALSE;
   S707_LM_DC_2ND_CLAMP1.Visu_Ret_Arr[10] := FALSE;
   S707_LM_DC_2ND_CLAMP1.Visu_Ret_Arr[11] := FALSE;
   S707_LM_DC_2ND_CLAMP1.Visu_Ret_Arr[12] := FALSE;
   S707_LM_DC_2ND_CLAMP1.Visu_Ret_Arr[13] := FALSE;
   S707_LM_DC_2ND_CLAMP1.Visu_Ret_Arr[14] := FALSE;
   S707_LM_DC_2ND_CLAMP1.Visu_Ret_Arr[15] := FALSE;
   S707_LM_DC_2ND_CLAMP1.BLK_Move_Ret := 0;
   S707_LM_DC_2ND_CLAMP1.Enable := FALSE;
   S707_LM_DC_2ND_CLAMP1.Adv_End := FALSE;
   S707_LM_DC_2ND_CLAMP1.Ret_End := FALSE;
   S707_LM_DC_2ND_CLAMP2.Enable_Aux := FALSE;
   S707_LM_DC_2ND_CLAMP2.Adv_Amount := 1;
   S707_LM_DC_2ND_CLAMP2.Ret_Amount := 1;
   S707_LM_DC_2ND_CLAMP2.LS_Adv1 := FALSE;
   S707_LM_DC_2ND_CLAMP2.LS_Ret1 := FALSE;
   S707_LM_DC_2ND_CLAMP2.LS_Adv2 := FALSE;
   S707_LM_DC_2ND_CLAMP2.LS_Ret2 := FALSE;
   S707_LM_DC_2ND_CLAMP2.LS_Adv3 := FALSE;
   S707_LM_DC_2ND_CLAMP2.LS_Ret3 := FALSE;
   S707_LM_DC_2ND_CLAMP2.LS_Adv4 := FALSE;
   S707_LM_DC_2ND_CLAMP2.LS_Ret4 := FALSE;
   S707_LM_DC_2ND_CLAMP2.SOL_Adv := FALSE;
   S707_LM_DC_2ND_CLAMP2.SOL_Ret := FALSE;
   S707_LM_DC_2ND_CLAMP2.M_Ready := TRUE;
   S707_LM_DC_2ND_CLAMP2.T_CHK1 := T#4S;
   S707_LM_DC_2ND_CLAMP2.T_CHK2 := T#4S;
   S707_LM_DC_2ND_CLAMP2.PB_Lamp_CHK := FALSE;
   S707_LM_DC_2ND_CLAMP2.PB_Error_Rst := FALSE;
   S707_LM_DC_2ND_CLAMP2.M_FLICK := TRUE;
   S707_LM_DC_2ND_CLAMP2.M_Adv_Err := FALSE;
   S707_LM_DC_2ND_CLAMP2.M_Ret_Err := FALSE;
   S707_LM_DC_2ND_CLAMP2.LP_Adv := FALSE;
   S707_LM_DC_2ND_CLAMP2.LP_Ret := FALSE;
   S707_LM_DC_2ND_CLAMP2.Visu_Adv := W#16#0;
   S707_LM_DC_2ND_CLAMP2.Visu_Ret := W#16#0;
   S707_LM_DC_2ND_CLAMP2.Error_T1.IN := FALSE;
   S707_LM_DC_2ND_CLAMP2.Error_T1.PT := T#4S;
   S707_LM_DC_2ND_CLAMP2.Error_T1.Q := FALSE;
   S707_LM_DC_2ND_CLAMP2.Error_T1.ET := T#0MS;
   S707_LM_DC_2ND_CLAMP2.Error_T1.STATE := B#16#0;
   S707_LM_DC_2ND_CLAMP2.Error_T1.STIME := T#0MS;
   S707_LM_DC_2ND_CLAMP2.Error_T1.ATIME := T#0MS;
   S707_LM_DC_2ND_CLAMP2.Error_T2.IN := FALSE;
   S707_LM_DC_2ND_CLAMP2.Error_T2.PT := T#4S;
   S707_LM_DC_2ND_CLAMP2.Error_T2.Q := FALSE;
   S707_LM_DC_2ND_CLAMP2.Error_T2.ET := T#0MS;
   S707_LM_DC_2ND_CLAMP2.Error_T2.STATE := B#16#0;
   S707_LM_DC_2ND_CLAMP2.Error_T2.STIME := T#0MS;
   S707_LM_DC_2ND_CLAMP2.Error_T2.ATIME := T#0MS;
   S707_LM_DC_2ND_CLAMP2.CHK_Aux1 := FALSE;
   S707_LM_DC_2ND_CLAMP2.CHK_Aux2 := FALSE;
   S707_LM_DC_2ND_CLAMP2.Error_T1_DN := FALSE;
   S707_LM_DC_2ND_CLAMP2.Error_T2_DN := FALSE;
   S707_LM_DC_2ND_CLAMP2.Adv_Memo := TRUE;
   S707_LM_DC_2ND_CLAMP2.Visu_Adv_Arr[0] := FALSE;
   S707_LM_DC_2ND_CLAMP2.Visu_Adv_Arr[1] := FALSE;
   S707_LM_DC_2ND_CLAMP2.Visu_Adv_Arr[2] := FALSE;
   S707_LM_DC_2ND_CLAMP2.Visu_Adv_Arr[3] := FALSE;
   S707_LM_DC_2ND_CLAMP2.Visu_Adv_Arr[4] := FALSE;
   S707_LM_DC_2ND_CLAMP2.Visu_Adv_Arr[5] := FALSE;
   S707_LM_DC_2ND_CLAMP2.Visu_Adv_Arr[6] := FALSE;
   S707_LM_DC_2ND_CLAMP2.Visu_Adv_Arr[7] := FALSE;
   S707_LM_DC_2ND_CLAMP2.Visu_Adv_Arr[8] := FALSE;
   S707_LM_DC_2ND_CLAMP2.Visu_Adv_Arr[9] := FALSE;
   S707_LM_DC_2ND_CLAMP2.Visu_Adv_Arr[10] := FALSE;
   S707_LM_DC_2ND_CLAMP2.Visu_Adv_Arr[11] := FALSE;
   S707_LM_DC_2ND_CLAMP2.Visu_Adv_Arr[12] := FALSE;
   S707_LM_DC_2ND_CLAMP2.Visu_Adv_Arr[13] := FALSE;
   S707_LM_DC_2ND_CLAMP2.Visu_Adv_Arr[14] := FALSE;
   S707_LM_DC_2ND_CLAMP2.Visu_Adv_Arr[15] := FALSE;
   S707_LM_DC_2ND_CLAMP2.Visu_Ret_Arr[0] := FALSE;
   S707_LM_DC_2ND_CLAMP2.Visu_Ret_Arr[1] := FALSE;
   S707_LM_DC_2ND_CLAMP2.Visu_Ret_Arr[2] := FALSE;
   S707_LM_DC_2ND_CLAMP2.Visu_Ret_Arr[3] := FALSE;
   S707_LM_DC_2ND_CLAMP2.Visu_Ret_Arr[4] := FALSE;
   S707_LM_DC_2ND_CLAMP2.Visu_Ret_Arr[5] := FALSE;
   S707_LM_DC_2ND_CLAMP2.Visu_Ret_Arr[6] := FALSE;
   S707_LM_DC_2ND_CLAMP2.Visu_Ret_Arr[7] := FALSE;
   S707_LM_DC_2ND_CLAMP2.Visu_Ret_Arr[8] := FALSE;
   S707_LM_DC_2ND_CLAMP2.Visu_Ret_Arr[9] := FALSE;
   S707_LM_DC_2ND_CLAMP2.Visu_Ret_Arr[10] := FALSE;
   S707_LM_DC_2ND_CLAMP2.Visu_Ret_Arr[11] := FALSE;
   S707_LM_DC_2ND_CLAMP2.Visu_Ret_Arr[12] := FALSE;
   S707_LM_DC_2ND_CLAMP2.Visu_Ret_Arr[13] := FALSE;
   S707_LM_DC_2ND_CLAMP2.Visu_Ret_Arr[14] := FALSE;
   S707_LM_DC_2ND_CLAMP2.Visu_Ret_Arr[15] := FALSE;
   S707_LM_DC_2ND_CLAMP2.BLK_Move_Ret := 0;
   S707_LM_DC_2ND_CLAMP2.Enable := FALSE;
   S707_LM_DC_2ND_CLAMP2.Adv_End := FALSE;
   S707_LM_DC_2ND_CLAMP2.Ret_End := FALSE;
   S707_LM_DC_2ND_CLAMP3.Enable_Aux := FALSE;
   S707_LM_DC_2ND_CLAMP3.Adv_Amount := 1;
   S707_LM_DC_2ND_CLAMP3.Ret_Amount := 1;
   S707_LM_DC_2ND_CLAMP3.LS_Adv1 := FALSE;
   S707_LM_DC_2ND_CLAMP3.LS_Ret1 := FALSE;
   S707_LM_DC_2ND_CLAMP3.LS_Adv2 := FALSE;
   S707_LM_DC_2ND_CLAMP3.LS_Ret2 := FALSE;
   S707_LM_DC_2ND_CLAMP3.LS_Adv3 := FALSE;
   S707_LM_DC_2ND_CLAMP3.LS_Ret3 := FALSE;
   S707_LM_DC_2ND_CLAMP3.LS_Adv4 := FALSE;
   S707_LM_DC_2ND_CLAMP3.LS_Ret4 := FALSE;
   S707_LM_DC_2ND_CLAMP3.SOL_Adv := FALSE;
   S707_LM_DC_2ND_CLAMP3.SOL_Ret := FALSE;
   S707_LM_DC_2ND_CLAMP3.M_Ready := TRUE;
   S707_LM_DC_2ND_CLAMP3.T_CHK1 := T#4S;
   S707_LM_DC_2ND_CLAMP3.T_CHK2 := T#4S;
   S707_LM_DC_2ND_CLAMP3.PB_Lamp_CHK := FALSE;
   S707_LM_DC_2ND_CLAMP3.PB_Error_Rst := FALSE;
   S707_LM_DC_2ND_CLAMP3.M_FLICK := TRUE;
   S707_LM_DC_2ND_CLAMP3.M_Adv_Err := FALSE;
   S707_LM_DC_2ND_CLAMP3.M_Ret_Err := FALSE;
   S707_LM_DC_2ND_CLAMP3.LP_Adv := FALSE;
   S707_LM_DC_2ND_CLAMP3.LP_Ret := FALSE;
   S707_LM_DC_2ND_CLAMP3.Visu_Adv := W#16#0;
   S707_LM_DC_2ND_CLAMP3.Visu_Ret := W#16#0;
   S707_LM_DC_2ND_CLAMP3.Error_T1.IN := FALSE;
   S707_LM_DC_2ND_CLAMP3.Error_T1.PT := T#4S;
   S707_LM_DC_2ND_CLAMP3.Error_T1.Q := FALSE;
   S707_LM_DC_2ND_CLAMP3.Error_T1.ET := T#0MS;
   S707_LM_DC_2ND_CLAMP3.Error_T1.STATE := B#16#0;
   S707_LM_DC_2ND_CLAMP3.Error_T1.STIME := T#0MS;
   S707_LM_DC_2ND_CLAMP3.Error_T1.ATIME := T#0MS;
   S707_LM_DC_2ND_CLAMP3.Error_T2.IN := FALSE;
   S707_LM_DC_2ND_CLAMP3.Error_T2.PT := T#4S;
   S707_LM_DC_2ND_CLAMP3.Error_T2.Q := FALSE;
   S707_LM_DC_2ND_CLAMP3.Error_T2.ET := T#0MS;
   S707_LM_DC_2ND_CLAMP3.Error_T2.STATE := B#16#0;
   S707_LM_DC_2ND_CLAMP3.Error_T2.STIME := T#0MS;
   S707_LM_DC_2ND_CLAMP3.Error_T2.ATIME := T#0MS;
   S707_LM_DC_2ND_CLAMP3.CHK_Aux1 := FALSE;
   S707_LM_DC_2ND_CLAMP3.CHK_Aux2 := FALSE;
   S707_LM_DC_2ND_CLAMP3.Error_T1_DN := FALSE;
   S707_LM_DC_2ND_CLAMP3.Error_T2_DN := FALSE;
   S707_LM_DC_2ND_CLAMP3.Adv_Memo := TRUE;
   S707_LM_DC_2ND_CLAMP3.Visu_Adv_Arr[0] := FALSE;
   S707_LM_DC_2ND_CLAMP3.Visu_Adv_Arr[1] := FALSE;
   S707_LM_DC_2ND_CLAMP3.Visu_Adv_Arr[2] := FALSE;
   S707_LM_DC_2ND_CLAMP3.Visu_Adv_Arr[3] := FALSE;
   S707_LM_DC_2ND_CLAMP3.Visu_Adv_Arr[4] := FALSE;
   S707_LM_DC_2ND_CLAMP3.Visu_Adv_Arr[5] := FALSE;
   S707_LM_DC_2ND_CLAMP3.Visu_Adv_Arr[6] := FALSE;
   S707_LM_DC_2ND_CLAMP3.Visu_Adv_Arr[7] := FALSE;
   S707_LM_DC_2ND_CLAMP3.Visu_Adv_Arr[8] := FALSE;
   S707_LM_DC_2ND_CLAMP3.Visu_Adv_Arr[9] := FALSE;
   S707_LM_DC_2ND_CLAMP3.Visu_Adv_Arr[10] := FALSE;
   S707_LM_DC_2ND_CLAMP3.Visu_Adv_Arr[11] := FALSE;
   S707_LM_DC_2ND_CLAMP3.Visu_Adv_Arr[12] := FALSE;
   S707_LM_DC_2ND_CLAMP3.Visu_Adv_Arr[13] := FALSE;
   S707_LM_DC_2ND_CLAMP3.Visu_Adv_Arr[14] := FALSE;
   S707_LM_DC_2ND_CLAMP3.Visu_Adv_Arr[15] := FALSE;
   S707_LM_DC_2ND_CLAMP3.Visu_Ret_Arr[0] := FALSE;
   S707_LM_DC_2ND_CLAMP3.Visu_Ret_Arr[1] := FALSE;
   S707_LM_DC_2ND_CLAMP3.Visu_Ret_Arr[2] := FALSE;
   S707_LM_DC_2ND_CLAMP3.Visu_Ret_Arr[3] := FALSE;
   S707_LM_DC_2ND_CLAMP3.Visu_Ret_Arr[4] := FALSE;
   S707_LM_DC_2ND_CLAMP3.Visu_Ret_Arr[5] := FALSE;
   S707_LM_DC_2ND_CLAMP3.Visu_Ret_Arr[6] := FALSE;
   S707_LM_DC_2ND_CLAMP3.Visu_Ret_Arr[7] := FALSE;
   S707_LM_DC_2ND_CLAMP3.Visu_Ret_Arr[8] := FALSE;
   S707_LM_DC_2ND_CLAMP3.Visu_Ret_Arr[9] := FALSE;
   S707_LM_DC_2ND_CLAMP3.Visu_Ret_Arr[10] := FALSE;
   S707_LM_DC_2ND_CLAMP3.Visu_Ret_Arr[11] := FALSE;
   S707_LM_DC_2ND_CLAMP3.Visu_Ret_Arr[12] := FALSE;
   S707_LM_DC_2ND_CLAMP3.Visu_Ret_Arr[13] := FALSE;
   S707_LM_DC_2ND_CLAMP3.Visu_Ret_Arr[14] := FALSE;
   S707_LM_DC_2ND_CLAMP3.Visu_Ret_Arr[15] := FALSE;
   S707_LM_DC_2ND_CLAMP3.BLK_Move_Ret := 0;
   S707_LM_DC_2ND_CLAMP3.Enable := FALSE;
   S707_LM_DC_2ND_CLAMP3.Adv_End := FALSE;
   S707_LM_DC_2ND_CLAMP3.Ret_End := FALSE;
   S707_LM_DC_2ND_CLAMP4.Enable_Aux := FALSE;
   S707_LM_DC_2ND_CLAMP4.Adv_Amount := 1;
   S707_LM_DC_2ND_CLAMP4.Ret_Amount := 1;
   S707_LM_DC_2ND_CLAMP4.LS_Adv1 := FALSE;
   S707_LM_DC_2ND_CLAMP4.LS_Ret1 := FALSE;
   S707_LM_DC_2ND_CLAMP4.LS_Adv2 := FALSE;
   S707_LM_DC_2ND_CLAMP4.LS_Ret2 := FALSE;
   S707_LM_DC_2ND_CLAMP4.LS_Adv3 := FALSE;
   S707_LM_DC_2ND_CLAMP4.LS_Ret3 := FALSE;
   S707_LM_DC_2ND_CLAMP4.LS_Adv4 := FALSE;
   S707_LM_DC_2ND_CLAMP4.LS_Ret4 := FALSE;
   S707_LM_DC_2ND_CLAMP4.SOL_Adv := FALSE;
   S707_LM_DC_2ND_CLAMP4.SOL_Ret := FALSE;
   S707_LM_DC_2ND_CLAMP4.M_Ready := TRUE;
   S707_LM_DC_2ND_CLAMP4.T_CHK1 := T#4S;
   S707_LM_DC_2ND_CLAMP4.T_CHK2 := T#4S;
   S707_LM_DC_2ND_CLAMP4.PB_Lamp_CHK := FALSE;
   S707_LM_DC_2ND_CLAMP4.PB_Error_Rst := FALSE;
   S707_LM_DC_2ND_CLAMP4.M_FLICK := TRUE;
   S707_LM_DC_2ND_CLAMP4.M_Adv_Err := FALSE;
   S707_LM_DC_2ND_CLAMP4.M_Ret_Err := FALSE;
   S707_LM_DC_2ND_CLAMP4.LP_Adv := FALSE;
   S707_LM_DC_2ND_CLAMP4.LP_Ret := FALSE;
   S707_LM_DC_2ND_CLAMP4.Visu_Adv := W#16#0;
   S707_LM_DC_2ND_CLAMP4.Visu_Ret := W#16#0;
   S707_LM_DC_2ND_CLAMP4.Error_T1.IN := FALSE;
   S707_LM_DC_2ND_CLAMP4.Error_T1.PT := T#4S;
   S707_LM_DC_2ND_CLAMP4.Error_T1.Q := FALSE;
   S707_LM_DC_2ND_CLAMP4.Error_T1.ET := T#0MS;
   S707_LM_DC_2ND_CLAMP4.Error_T1.STATE := B#16#0;
   S707_LM_DC_2ND_CLAMP4.Error_T1.STIME := T#0MS;
   S707_LM_DC_2ND_CLAMP4.Error_T1.ATIME := T#0MS;
   S707_LM_DC_2ND_CLAMP4.Error_T2.IN := FALSE;
   S707_LM_DC_2ND_CLAMP4.Error_T2.PT := T#4S;
   S707_LM_DC_2ND_CLAMP4.Error_T2.Q := FALSE;
   S707_LM_DC_2ND_CLAMP4.Error_T2.ET := T#0MS;
   S707_LM_DC_2ND_CLAMP4.Error_T2.STATE := B#16#0;
   S707_LM_DC_2ND_CLAMP4.Error_T2.STIME := T#0MS;
   S707_LM_DC_2ND_CLAMP4.Error_T2.ATIME := T#0MS;
   S707_LM_DC_2ND_CLAMP4.CHK_Aux1 := FALSE;
   S707_LM_DC_2ND_CLAMP4.CHK_Aux2 := FALSE;
   S707_LM_DC_2ND_CLAMP4.Error_T1_DN := FALSE;
   S707_LM_DC_2ND_CLAMP4.Error_T2_DN := FALSE;
   S707_LM_DC_2ND_CLAMP4.Adv_Memo := FALSE;
   S707_LM_DC_2ND_CLAMP4.Visu_Adv_Arr[0] := FALSE;
   S707_LM_DC_2ND_CLAMP4.Visu_Adv_Arr[1] := FALSE;
   S707_LM_DC_2ND_CLAMP4.Visu_Adv_Arr[2] := FALSE;
   S707_LM_DC_2ND_CLAMP4.Visu_Adv_Arr[3] := FALSE;
   S707_LM_DC_2ND_CLAMP4.Visu_Adv_Arr[4] := FALSE;
   S707_LM_DC_2ND_CLAMP4.Visu_Adv_Arr[5] := FALSE;
   S707_LM_DC_2ND_CLAMP4.Visu_Adv_Arr[6] := FALSE;
   S707_LM_DC_2ND_CLAMP4.Visu_Adv_Arr[7] := FALSE;
   S707_LM_DC_2ND_CLAMP4.Visu_Adv_Arr[8] := FALSE;
   S707_LM_DC_2ND_CLAMP4.Visu_Adv_Arr[9] := FALSE;
   S707_LM_DC_2ND_CLAMP4.Visu_Adv_Arr[10] := FALSE;
   S707_LM_DC_2ND_CLAMP4.Visu_Adv_Arr[11] := FALSE;
   S707_LM_DC_2ND_CLAMP4.Visu_Adv_Arr[12] := FALSE;
   S707_LM_DC_2ND_CLAMP4.Visu_Adv_Arr[13] := FALSE;
   S707_LM_DC_2ND_CLAMP4.Visu_Adv_Arr[14] := FALSE;
   S707_LM_DC_2ND_CLAMP4.Visu_Adv_Arr[15] := FALSE;
   S707_LM_DC_2ND_CLAMP4.Visu_Ret_Arr[0] := FALSE;
   S707_LM_DC_2ND_CLAMP4.Visu_Ret_Arr[1] := FALSE;
   S707_LM_DC_2ND_CLAMP4.Visu_Ret_Arr[2] := FALSE;
   S707_LM_DC_2ND_CLAMP4.Visu_Ret_Arr[3] := FALSE;
   S707_LM_DC_2ND_CLAMP4.Visu_Ret_Arr[4] := FALSE;
   S707_LM_DC_2ND_CLAMP4.Visu_Ret_Arr[5] := FALSE;
   S707_LM_DC_2ND_CLAMP4.Visu_Ret_Arr[6] := FALSE;
   S707_LM_DC_2ND_CLAMP4.Visu_Ret_Arr[7] := FALSE;
   S707_LM_DC_2ND_CLAMP4.Visu_Ret_Arr[8] := FALSE;
   S707_LM_DC_2ND_CLAMP4.Visu_Ret_Arr[9] := FALSE;
   S707_LM_DC_2ND_CLAMP4.Visu_Ret_Arr[10] := FALSE;
   S707_LM_DC_2ND_CLAMP4.Visu_Ret_Arr[11] := FALSE;
   S707_LM_DC_2ND_CLAMP4.Visu_Ret_Arr[12] := FALSE;
   S707_LM_DC_2ND_CLAMP4.Visu_Ret_Arr[13] := FALSE;
   S707_LM_DC_2ND_CLAMP4.Visu_Ret_Arr[14] := FALSE;
   S707_LM_DC_2ND_CLAMP4.Visu_Ret_Arr[15] := FALSE;
   S707_LM_DC_2ND_CLAMP4.BLK_Move_Ret := 0;
   S707_LM_DC_2ND_CLAMP4.Enable := FALSE;
   S707_LM_DC_2ND_CLAMP4.Adv_End := FALSE;
   S707_LM_DC_2ND_CLAMP4.Ret_End := FALSE;
   S707_LM_DC_2ND_CLAMP5.Enable_Aux := FALSE;
   S707_LM_DC_2ND_CLAMP5.Adv_Amount := 1;
   S707_LM_DC_2ND_CLAMP5.Ret_Amount := 1;
   S707_LM_DC_2ND_CLAMP5.LS_Adv1 := FALSE;
   S707_LM_DC_2ND_CLAMP5.LS_Ret1 := FALSE;
   S707_LM_DC_2ND_CLAMP5.LS_Adv2 := FALSE;
   S707_LM_DC_2ND_CLAMP5.LS_Ret2 := FALSE;
   S707_LM_DC_2ND_CLAMP5.LS_Adv3 := FALSE;
   S707_LM_DC_2ND_CLAMP5.LS_Ret3 := FALSE;
   S707_LM_DC_2ND_CLAMP5.LS_Adv4 := FALSE;
   S707_LM_DC_2ND_CLAMP5.LS_Ret4 := FALSE;
   S707_LM_DC_2ND_CLAMP5.SOL_Adv := FALSE;
   S707_LM_DC_2ND_CLAMP5.SOL_Ret := FALSE;
   S707_LM_DC_2ND_CLAMP5.M_Ready := TRUE;
   S707_LM_DC_2ND_CLAMP5.T_CHK1 := T#4S;
   S707_LM_DC_2ND_CLAMP5.T_CHK2 := T#4S;
   S707_LM_DC_2ND_CLAMP5.PB_Lamp_CHK := FALSE;
   S707_LM_DC_2ND_CLAMP5.PB_Error_Rst := FALSE;
   S707_LM_DC_2ND_CLAMP5.M_FLICK := TRUE;
   S707_LM_DC_2ND_CLAMP5.M_Adv_Err := FALSE;
   S707_LM_DC_2ND_CLAMP5.M_Ret_Err := FALSE;
   S707_LM_DC_2ND_CLAMP5.LP_Adv := FALSE;
   S707_LM_DC_2ND_CLAMP5.LP_Ret := FALSE;
   S707_LM_DC_2ND_CLAMP5.Visu_Adv := W#16#0;
   S707_LM_DC_2ND_CLAMP5.Visu_Ret := W#16#0;
   S707_LM_DC_2ND_CLAMP5.Error_T1.IN := FALSE;
   S707_LM_DC_2ND_CLAMP5.Error_T1.PT := T#4S;
   S707_LM_DC_2ND_CLAMP5.Error_T1.Q := FALSE;
   S707_LM_DC_2ND_CLAMP5.Error_T1.ET := T#0MS;
   S707_LM_DC_2ND_CLAMP5.Error_T1.STATE := B#16#0;
   S707_LM_DC_2ND_CLAMP5.Error_T1.STIME := T#0MS;
   S707_LM_DC_2ND_CLAMP5.Error_T1.ATIME := T#0MS;
   S707_LM_DC_2ND_CLAMP5.Error_T2.IN := FALSE;
   S707_LM_DC_2ND_CLAMP5.Error_T2.PT := T#4S;
   S707_LM_DC_2ND_CLAMP5.Error_T2.Q := FALSE;
   S707_LM_DC_2ND_CLAMP5.Error_T2.ET := T#0MS;
   S707_LM_DC_2ND_CLAMP5.Error_T2.STATE := B#16#0;
   S707_LM_DC_2ND_CLAMP5.Error_T2.STIME := T#0MS;
   S707_LM_DC_2ND_CLAMP5.Error_T2.ATIME := T#0MS;
   S707_LM_DC_2ND_CLAMP5.CHK_Aux1 := FALSE;
   S707_LM_DC_2ND_CLAMP5.CHK_Aux2 := FALSE;
   S707_LM_DC_2ND_CLAMP5.Error_T1_DN := FALSE;
   S707_LM_DC_2ND_CLAMP5.Error_T2_DN := FALSE;
   S707_LM_DC_2ND_CLAMP5.Adv_Memo := FALSE;
   S707_LM_DC_2ND_CLAMP5.Visu_Adv_Arr[0] := FALSE;
   S707_LM_DC_2ND_CLAMP5.Visu_Adv_Arr[1] := FALSE;
   S707_LM_DC_2ND_CLAMP5.Visu_Adv_Arr[2] := FALSE;
   S707_LM_DC_2ND_CLAMP5.Visu_Adv_Arr[3] := FALSE;
   S707_LM_DC_2ND_CLAMP5.Visu_Adv_Arr[4] := FALSE;
   S707_LM_DC_2ND_CLAMP5.Visu_Adv_Arr[5] := FALSE;
   S707_LM_DC_2ND_CLAMP5.Visu_Adv_Arr[6] := FALSE;
   S707_LM_DC_2ND_CLAMP5.Visu_Adv_Arr[7] := FALSE;
   S707_LM_DC_2ND_CLAMP5.Visu_Adv_Arr[8] := FALSE;
   S707_LM_DC_2ND_CLAMP5.Visu_Adv_Arr[9] := FALSE;
   S707_LM_DC_2ND_CLAMP5.Visu_Adv_Arr[10] := FALSE;
   S707_LM_DC_2ND_CLAMP5.Visu_Adv_Arr[11] := FALSE;
   S707_LM_DC_2ND_CLAMP5.Visu_Adv_Arr[12] := FALSE;
   S707_LM_DC_2ND_CLAMP5.Visu_Adv_Arr[13] := FALSE;
   S707_LM_DC_2ND_CLAMP5.Visu_Adv_Arr[14] := FALSE;
   S707_LM_DC_2ND_CLAMP5.Visu_Adv_Arr[15] := FALSE;
   S707_LM_DC_2ND_CLAMP5.Visu_Ret_Arr[0] := FALSE;
   S707_LM_DC_2ND_CLAMP5.Visu_Ret_Arr[1] := FALSE;
   S707_LM_DC_2ND_CLAMP5.Visu_Ret_Arr[2] := FALSE;
   S707_LM_DC_2ND_CLAMP5.Visu_Ret_Arr[3] := FALSE;
   S707_LM_DC_2ND_CLAMP5.Visu_Ret_Arr[4] := FALSE;
   S707_LM_DC_2ND_CLAMP5.Visu_Ret_Arr[5] := FALSE;
   S707_LM_DC_2ND_CLAMP5.Visu_Ret_Arr[6] := FALSE;
   S707_LM_DC_2ND_CLAMP5.Visu_Ret_Arr[7] := FALSE;
   S707_LM_DC_2ND_CLAMP5.Visu_Ret_Arr[8] := FALSE;
   S707_LM_DC_2ND_CLAMP5.Visu_Ret_Arr[9] := FALSE;
   S707_LM_DC_2ND_CLAMP5.Visu_Ret_Arr[10] := FALSE;
   S707_LM_DC_2ND_CLAMP5.Visu_Ret_Arr[11] := FALSE;
   S707_LM_DC_2ND_CLAMP5.Visu_Ret_Arr[12] := FALSE;
   S707_LM_DC_2ND_CLAMP5.Visu_Ret_Arr[13] := FALSE;
   S707_LM_DC_2ND_CLAMP5.Visu_Ret_Arr[14] := FALSE;
   S707_LM_DC_2ND_CLAMP5.Visu_Ret_Arr[15] := FALSE;
   S707_LM_DC_2ND_CLAMP5.BLK_Move_Ret := 0;
   S707_LM_DC_2ND_CLAMP5.Enable := FALSE;
   S707_LM_DC_2ND_CLAMP5.Adv_End := FALSE;
   S707_LM_DC_2ND_CLAMP5.Ret_End := FALSE;
   S707_LM_DC_STK_PIN.Enable_Aux := FALSE;
   S707_LM_DC_STK_PIN.Adv_Amount := 1;
   S707_LM_DC_STK_PIN.Ret_Amount := 1;
   S707_LM_DC_STK_PIN.LS_Adv1 := FALSE;
   S707_LM_DC_STK_PIN.LS_Ret1 := FALSE;
   S707_LM_DC_STK_PIN.LS_Adv2 := FALSE;
   S707_LM_DC_STK_PIN.LS_Ret2 := FALSE;
   S707_LM_DC_STK_PIN.LS_Adv3 := FALSE;
   S707_LM_DC_STK_PIN.LS_Ret3 := FALSE;
   S707_LM_DC_STK_PIN.LS_Adv4 := FALSE;
   S707_LM_DC_STK_PIN.LS_Ret4 := FALSE;
   S707_LM_DC_STK_PIN.SOL_Adv := FALSE;
   S707_LM_DC_STK_PIN.SOL_Ret := FALSE;
   S707_LM_DC_STK_PIN.M_Ready := TRUE;
   S707_LM_DC_STK_PIN.T_CHK1 := T#4S;
   S707_LM_DC_STK_PIN.T_CHK2 := T#4S;
   S707_LM_DC_STK_PIN.PB_Lamp_CHK := FALSE;
   S707_LM_DC_STK_PIN.PB_Error_Rst := FALSE;
   S707_LM_DC_STK_PIN.M_FLICK := TRUE;
   S707_LM_DC_STK_PIN.M_Adv_Err := FALSE;
   S707_LM_DC_STK_PIN.M_Ret_Err := FALSE;
   S707_LM_DC_STK_PIN.LP_Adv := FALSE;
   S707_LM_DC_STK_PIN.LP_Ret := FALSE;
   S707_LM_DC_STK_PIN.Visu_Adv := W#16#0;
   S707_LM_DC_STK_PIN.Visu_Ret := W#16#0;
   S707_LM_DC_STK_PIN.Error_T1.IN := FALSE;
   S707_LM_DC_STK_PIN.Error_T1.PT := T#4S;
   S707_LM_DC_STK_PIN.Error_T1.Q := FALSE;
   S707_LM_DC_STK_PIN.Error_T1.ET := T#0MS;
   S707_LM_DC_STK_PIN.Error_T1.STATE := B#16#0;
   S707_LM_DC_STK_PIN.Error_T1.STIME := T#15D12H51M13S521MS;
   S707_LM_DC_STK_PIN.Error_T1.ATIME := T#15D12H51M13S927MS;
   S707_LM_DC_STK_PIN.Error_T2.IN := FALSE;
   S707_LM_DC_STK_PIN.Error_T2.PT := T#4S;
   S707_LM_DC_STK_PIN.Error_T2.Q := FALSE;
   S707_LM_DC_STK_PIN.Error_T2.ET := T#0MS;
   S707_LM_DC_STK_PIN.Error_T2.STATE := B#16#0;
   S707_LM_DC_STK_PIN.Error_T2.STIME := T#0MS;
   S707_LM_DC_STK_PIN.Error_T2.ATIME := T#0MS;
   S707_LM_DC_STK_PIN.CHK_Aux1 := FALSE;
   S707_LM_DC_STK_PIN.CHK_Aux2 := FALSE;
   S707_LM_DC_STK_PIN.Error_T1_DN := FALSE;
   S707_LM_DC_STK_PIN.Error_T2_DN := FALSE;
   S707_LM_DC_STK_PIN.Adv_Memo := FALSE;
   S707_LM_DC_STK_PIN.Visu_Adv_Arr[0] := FALSE;
   S707_LM_DC_STK_PIN.Visu_Adv_Arr[1] := FALSE;
   S707_LM_DC_STK_PIN.Visu_Adv_Arr[2] := FALSE;
   S707_LM_DC_STK_PIN.Visu_Adv_Arr[3] := FALSE;
   S707_LM_DC_STK_PIN.Visu_Adv_Arr[4] := FALSE;
   S707_LM_DC_STK_PIN.Visu_Adv_Arr[5] := FALSE;
   S707_LM_DC_STK_PIN.Visu_Adv_Arr[6] := FALSE;
   S707_LM_DC_STK_PIN.Visu_Adv_Arr[7] := FALSE;
   S707_LM_DC_STK_PIN.Visu_Adv_Arr[8] := FALSE;
   S707_LM_DC_STK_PIN.Visu_Adv_Arr[9] := FALSE;
   S707_LM_DC_STK_PIN.Visu_Adv_Arr[10] := FALSE;
   S707_LM_DC_STK_PIN.Visu_Adv_Arr[11] := FALSE;
   S707_LM_DC_STK_PIN.Visu_Adv_Arr[12] := FALSE;
   S707_LM_DC_STK_PIN.Visu_Adv_Arr[13] := FALSE;
   S707_LM_DC_STK_PIN.Visu_Adv_Arr[14] := FALSE;
   S707_LM_DC_STK_PIN.Visu_Adv_Arr[15] := FALSE;
   S707_LM_DC_STK_PIN.Visu_Ret_Arr[0] := FALSE;
   S707_LM_DC_STK_PIN.Visu_Ret_Arr[1] := FALSE;
   S707_LM_DC_STK_PIN.Visu_Ret_Arr[2] := FALSE;
   S707_LM_DC_STK_PIN.Visu_Ret_Arr[3] := FALSE;
   S707_LM_DC_STK_PIN.Visu_Ret_Arr[4] := FALSE;
   S707_LM_DC_STK_PIN.Visu_Ret_Arr[5] := FALSE;
   S707_LM_DC_STK_PIN.Visu_Ret_Arr[6] := FALSE;
   S707_LM_DC_STK_PIN.Visu_Ret_Arr[7] := FALSE;
   S707_LM_DC_STK_PIN.Visu_Ret_Arr[8] := FALSE;
   S707_LM_DC_STK_PIN.Visu_Ret_Arr[9] := FALSE;
   S707_LM_DC_STK_PIN.Visu_Ret_Arr[10] := FALSE;
   S707_LM_DC_STK_PIN.Visu_Ret_Arr[11] := FALSE;
   S707_LM_DC_STK_PIN.Visu_Ret_Arr[12] := FALSE;
   S707_LM_DC_STK_PIN.Visu_Ret_Arr[13] := FALSE;
   S707_LM_DC_STK_PIN.Visu_Ret_Arr[14] := FALSE;
   S707_LM_DC_STK_PIN.Visu_Ret_Arr[15] := FALSE;
   S707_LM_DC_STK_PIN.BLK_Move_Ret := 0;
   S707_LM_DC_STK_PIN.Enable := FALSE;
   S707_LM_DC_STK_PIN.Adv_End := FALSE;
   S707_LM_DC_STK_PIN.Ret_End := FALSE;
   S707_LM_DC_OTR_CLAMP.Enable_Aux := FALSE;
   S707_LM_DC_OTR_CLAMP.Adv_Amount := 1;
   S707_LM_DC_OTR_CLAMP.Ret_Amount := 1;
   S707_LM_DC_OTR_CLAMP.LS_Adv1 := FALSE;
   S707_LM_DC_OTR_CLAMP.LS_Ret1 := FALSE;
   S707_LM_DC_OTR_CLAMP.LS_Adv2 := FALSE;
   S707_LM_DC_OTR_CLAMP.LS_Ret2 := FALSE;
   S707_LM_DC_OTR_CLAMP.LS_Adv3 := FALSE;
   S707_LM_DC_OTR_CLAMP.LS_Ret3 := FALSE;
   S707_LM_DC_OTR_CLAMP.LS_Adv4 := FALSE;
   S707_LM_DC_OTR_CLAMP.LS_Ret4 := FALSE;
   S707_LM_DC_OTR_CLAMP.SOL_Adv := FALSE;
   S707_LM_DC_OTR_CLAMP.SOL_Ret := FALSE;
   S707_LM_DC_OTR_CLAMP.M_Ready := TRUE;
   S707_LM_DC_OTR_CLAMP.T_CHK1 := T#4S;
   S707_LM_DC_OTR_CLAMP.T_CHK2 := T#4S;
   S707_LM_DC_OTR_CLAMP.PB_Lamp_CHK := FALSE;
   S707_LM_DC_OTR_CLAMP.PB_Error_Rst := FALSE;
   S707_LM_DC_OTR_CLAMP.M_FLICK := TRUE;
   S707_LM_DC_OTR_CLAMP.M_Adv_Err := FALSE;
   S707_LM_DC_OTR_CLAMP.M_Ret_Err := FALSE;
   S707_LM_DC_OTR_CLAMP.LP_Adv := FALSE;
   S707_LM_DC_OTR_CLAMP.LP_Ret := FALSE;
   S707_LM_DC_OTR_CLAMP.Visu_Adv := W#16#0;
   S707_LM_DC_OTR_CLAMP.Visu_Ret := W#16#0;
   S707_LM_DC_OTR_CLAMP.Error_T1.IN := FALSE;
   S707_LM_DC_OTR_CLAMP.Error_T1.PT := T#4S;
   S707_LM_DC_OTR_CLAMP.Error_T1.Q := FALSE;
   S707_LM_DC_OTR_CLAMP.Error_T1.ET := T#0MS;
   S707_LM_DC_OTR_CLAMP.Error_T1.STATE := B#16#0;
   S707_LM_DC_OTR_CLAMP.Error_T1.STIME := T#0MS;
   S707_LM_DC_OTR_CLAMP.Error_T1.ATIME := T#0MS;
   S707_LM_DC_OTR_CLAMP.Error_T2.IN := FALSE;
   S707_LM_DC_OTR_CLAMP.Error_T2.PT := T#4S;
   S707_LM_DC_OTR_CLAMP.Error_T2.Q := FALSE;
   S707_LM_DC_OTR_CLAMP.Error_T2.ET := T#0MS;
   S707_LM_DC_OTR_CLAMP.Error_T2.STATE := B#16#0;
   S707_LM_DC_OTR_CLAMP.Error_T2.STIME := T#0MS;
   S707_LM_DC_OTR_CLAMP.Error_T2.ATIME := T#0MS;
   S707_LM_DC_OTR_CLAMP.CHK_Aux1 := FALSE;
   S707_LM_DC_OTR_CLAMP.CHK_Aux2 := FALSE;
   S707_LM_DC_OTR_CLAMP.Error_T1_DN := FALSE;
   S707_LM_DC_OTR_CLAMP.Error_T2_DN := FALSE;
   S707_LM_DC_OTR_CLAMP.Adv_Memo := FALSE;
   S707_LM_DC_OTR_CLAMP.Visu_Adv_Arr[0] := FALSE;
   S707_LM_DC_OTR_CLAMP.Visu_Adv_Arr[1] := FALSE;
   S707_LM_DC_OTR_CLAMP.Visu_Adv_Arr[2] := FALSE;
   S707_LM_DC_OTR_CLAMP.Visu_Adv_Arr[3] := FALSE;
   S707_LM_DC_OTR_CLAMP.Visu_Adv_Arr[4] := FALSE;
   S707_LM_DC_OTR_CLAMP.Visu_Adv_Arr[5] := FALSE;
   S707_LM_DC_OTR_CLAMP.Visu_Adv_Arr[6] := FALSE;
   S707_LM_DC_OTR_CLAMP.Visu_Adv_Arr[7] := FALSE;
   S707_LM_DC_OTR_CLAMP.Visu_Adv_Arr[8] := FALSE;
   S707_LM_DC_OTR_CLAMP.Visu_Adv_Arr[9] := FALSE;
   S707_LM_DC_OTR_CLAMP.Visu_Adv_Arr[10] := FALSE;
   S707_LM_DC_OTR_CLAMP.Visu_Adv_Arr[11] := FALSE;
   S707_LM_DC_OTR_CLAMP.Visu_Adv_Arr[12] := FALSE;
   S707_LM_DC_OTR_CLAMP.Visu_Adv_Arr[13] := FALSE;
   S707_LM_DC_OTR_CLAMP.Visu_Adv_Arr[14] := FALSE;
   S707_LM_DC_OTR_CLAMP.Visu_Adv_Arr[15] := FALSE;
   S707_LM_DC_OTR_CLAMP.Visu_Ret_Arr[0] := FALSE;
   S707_LM_DC_OTR_CLAMP.Visu_Ret_Arr[1] := FALSE;
   S707_LM_DC_OTR_CLAMP.Visu_Ret_Arr[2] := FALSE;
   S707_LM_DC_OTR_CLAMP.Visu_Ret_Arr[3] := FALSE;
   S707_LM_DC_OTR_CLAMP.Visu_Ret_Arr[4] := FALSE;
   S707_LM_DC_OTR_CLAMP.Visu_Ret_Arr[5] := FALSE;
   S707_LM_DC_OTR_CLAMP.Visu_Ret_Arr[6] := FALSE;
   S707_LM_DC_OTR_CLAMP.Visu_Ret_Arr[7] := FALSE;
   S707_LM_DC_OTR_CLAMP.Visu_Ret_Arr[8] := FALSE;
   S707_LM_DC_OTR_CLAMP.Visu_Ret_Arr[9] := FALSE;
   S707_LM_DC_OTR_CLAMP.Visu_Ret_Arr[10] := FALSE;
   S707_LM_DC_OTR_CLAMP.Visu_Ret_Arr[11] := FALSE;
   S707_LM_DC_OTR_CLAMP.Visu_Ret_Arr[12] := FALSE;
   S707_LM_DC_OTR_CLAMP.Visu_Ret_Arr[13] := FALSE;
   S707_LM_DC_OTR_CLAMP.Visu_Ret_Arr[14] := FALSE;
   S707_LM_DC_OTR_CLAMP.Visu_Ret_Arr[15] := FALSE;
   S707_LM_DC_OTR_CLAMP.BLK_Move_Ret := 0;
   S707_LM_DC_OTR_CLAMP.Enable := FALSE;
   S707_LM_DC_OTR_CLAMP.Adv_End := FALSE;
   S707_LM_DC_OTR_CLAMP.Ret_End := FALSE;
   S707_LM_DC_ASSY_CLAMP.Enable_Aux := FALSE;
   S707_LM_DC_ASSY_CLAMP.Adv_Amount := 1;
   S707_LM_DC_ASSY_CLAMP.Ret_Amount := 1;
   S707_LM_DC_ASSY_CLAMP.LS_Adv1 := FALSE;
   S707_LM_DC_ASSY_CLAMP.LS_Ret1 := FALSE;
   S707_LM_DC_ASSY_CLAMP.LS_Adv2 := FALSE;
   S707_LM_DC_ASSY_CLAMP.LS_Ret2 := FALSE;
   S707_LM_DC_ASSY_CLAMP.LS_Adv3 := FALSE;
   S707_LM_DC_ASSY_CLAMP.LS_Ret3 := FALSE;
   S707_LM_DC_ASSY_CLAMP.LS_Adv4 := FALSE;
   S707_LM_DC_ASSY_CLAMP.LS_Ret4 := FALSE;
   S707_LM_DC_ASSY_CLAMP.SOL_Adv := FALSE;
   S707_LM_DC_ASSY_CLAMP.SOL_Ret := FALSE;
   S707_LM_DC_ASSY_CLAMP.M_Ready := TRUE;
   S707_LM_DC_ASSY_CLAMP.T_CHK1 := T#4S;
   S707_LM_DC_ASSY_CLAMP.T_CHK2 := T#4S;
   S707_LM_DC_ASSY_CLAMP.PB_Lamp_CHK := FALSE;
   S707_LM_DC_ASSY_CLAMP.PB_Error_Rst := FALSE;
   S707_LM_DC_ASSY_CLAMP.M_FLICK := TRUE;
   S707_LM_DC_ASSY_CLAMP.M_Adv_Err := FALSE;
   S707_LM_DC_ASSY_CLAMP.M_Ret_Err := FALSE;
   S707_LM_DC_ASSY_CLAMP.LP_Adv := FALSE;
   S707_LM_DC_ASSY_CLAMP.LP_Ret := FALSE;
   S707_LM_DC_ASSY_CLAMP.Visu_Adv := W#16#0;
   S707_LM_DC_ASSY_CLAMP.Visu_Ret := W#16#0;
   S707_LM_DC_ASSY_CLAMP.Error_T1.IN := FALSE;
   S707_LM_DC_ASSY_CLAMP.Error_T1.PT := T#4S;
   S707_LM_DC_ASSY_CLAMP.Error_T1.Q := FALSE;
   S707_LM_DC_ASSY_CLAMP.Error_T1.ET := T#0MS;
   S707_LM_DC_ASSY_CLAMP.Error_T1.STATE := B#16#0;
   S707_LM_DC_ASSY_CLAMP.Error_T1.STIME := T#0MS;
   S707_LM_DC_ASSY_CLAMP.Error_T1.ATIME := T#0MS;
   S707_LM_DC_ASSY_CLAMP.Error_T2.IN := FALSE;
   S707_LM_DC_ASSY_CLAMP.Error_T2.PT := T#4S;
   S707_LM_DC_ASSY_CLAMP.Error_T2.Q := FALSE;
   S707_LM_DC_ASSY_CLAMP.Error_T2.ET := T#0MS;
   S707_LM_DC_ASSY_CLAMP.Error_T2.STATE := B#16#0;
   S707_LM_DC_ASSY_CLAMP.Error_T2.STIME := T#0MS;
   S707_LM_DC_ASSY_CLAMP.Error_T2.ATIME := T#0MS;
   S707_LM_DC_ASSY_CLAMP.CHK_Aux1 := FALSE;
   S707_LM_DC_ASSY_CLAMP.CHK_Aux2 := FALSE;
   S707_LM_DC_ASSY_CLAMP.Error_T1_DN := FALSE;
   S707_LM_DC_ASSY_CLAMP.Error_T2_DN := FALSE;
   S707_LM_DC_ASSY_CLAMP.Adv_Memo := TRUE;
   S707_LM_DC_ASSY_CLAMP.Visu_Adv_Arr[0] := FALSE;
   S707_LM_DC_ASSY_CLAMP.Visu_Adv_Arr[1] := FALSE;
   S707_LM_DC_ASSY_CLAMP.Visu_Adv_Arr[2] := FALSE;
   S707_LM_DC_ASSY_CLAMP.Visu_Adv_Arr[3] := FALSE;
   S707_LM_DC_ASSY_CLAMP.Visu_Adv_Arr[4] := FALSE;
   S707_LM_DC_ASSY_CLAMP.Visu_Adv_Arr[5] := FALSE;
   S707_LM_DC_ASSY_CLAMP.Visu_Adv_Arr[6] := FALSE;
   S707_LM_DC_ASSY_CLAMP.Visu_Adv_Arr[7] := FALSE;
   S707_LM_DC_ASSY_CLAMP.Visu_Adv_Arr[8] := FALSE;
   S707_LM_DC_ASSY_CLAMP.Visu_Adv_Arr[9] := FALSE;
   S707_LM_DC_ASSY_CLAMP.Visu_Adv_Arr[10] := FALSE;
   S707_LM_DC_ASSY_CLAMP.Visu_Adv_Arr[11] := FALSE;
   S707_LM_DC_ASSY_CLAMP.Visu_Adv_Arr[12] := FALSE;
   S707_LM_DC_ASSY_CLAMP.Visu_Adv_Arr[13] := FALSE;
   S707_LM_DC_ASSY_CLAMP.Visu_Adv_Arr[14] := FALSE;
   S707_LM_DC_ASSY_CLAMP.Visu_Adv_Arr[15] := FALSE;
   S707_LM_DC_ASSY_CLAMP.Visu_Ret_Arr[0] := FALSE;
   S707_LM_DC_ASSY_CLAMP.Visu_Ret_Arr[1] := FALSE;
   S707_LM_DC_ASSY_CLAMP.Visu_Ret_Arr[2] := FALSE;
   S707_LM_DC_ASSY_CLAMP.Visu_Ret_Arr[3] := FALSE;
   S707_LM_DC_ASSY_CLAMP.Visu_Ret_Arr[4] := FALSE;
   S707_LM_DC_ASSY_CLAMP.Visu_Ret_Arr[5] := FALSE;
   S707_LM_DC_ASSY_CLAMP.Visu_Ret_Arr[6] := FALSE;
   S707_LM_DC_ASSY_CLAMP.Visu_Ret_Arr[7] := FALSE;
   S707_LM_DC_ASSY_CLAMP.Visu_Ret_Arr[8] := FALSE;
   S707_LM_DC_ASSY_CLAMP.Visu_Ret_Arr[9] := FALSE;
   S707_LM_DC_ASSY_CLAMP.Visu_Ret_Arr[10] := FALSE;
   S707_LM_DC_ASSY_CLAMP.Visu_Ret_Arr[11] := FALSE;
   S707_LM_DC_ASSY_CLAMP.Visu_Ret_Arr[12] := FALSE;
   S707_LM_DC_ASSY_CLAMP.Visu_Ret_Arr[13] := FALSE;
   S707_LM_DC_ASSY_CLAMP.Visu_Ret_Arr[14] := FALSE;
   S707_LM_DC_ASSY_CLAMP.Visu_Ret_Arr[15] := FALSE;
   S707_LM_DC_ASSY_CLAMP.BLK_Move_Ret := 0;
   S707_LM_DC_ASSY_CLAMP.Enable := FALSE;
   S707_LM_DC_ASSY_CLAMP.Adv_End := FALSE;
   S707_LM_DC_ASSY_CLAMP.Ret_End := FALSE;
   S707_LM_DC_FF_PIN.Enable_Aux := FALSE;
   S707_LM_DC_FF_PIN.Adv_Amount := 1;
   S707_LM_DC_FF_PIN.Ret_Amount := 1;
   S707_LM_DC_FF_PIN.LS_Adv1 := FALSE;
   S707_LM_DC_FF_PIN.LS_Ret1 := FALSE;
   S707_LM_DC_FF_PIN.LS_Adv2 := FALSE;
   S707_LM_DC_FF_PIN.LS_Ret2 := FALSE;
   S707_LM_DC_FF_PIN.LS_Adv3 := FALSE;
   S707_LM_DC_FF_PIN.LS_Ret3 := FALSE;
   S707_LM_DC_FF_PIN.LS_Adv4 := FALSE;
   S707_LM_DC_FF_PIN.LS_Ret4 := FALSE;
   S707_LM_DC_FF_PIN.SOL_Adv := FALSE;
   S707_LM_DC_FF_PIN.SOL_Ret := FALSE;
   S707_LM_DC_FF_PIN.M_Ready := TRUE;
   S707_LM_DC_FF_PIN.T_CHK1 := T#4S;
   S707_LM_DC_FF_PIN.T_CHK2 := T#4S;
   S707_LM_DC_FF_PIN.PB_Lamp_CHK := FALSE;
   S707_LM_DC_FF_PIN.PB_Error_Rst := FALSE;
   S707_LM_DC_FF_PIN.M_FLICK := TRUE;
   S707_LM_DC_FF_PIN.M_Adv_Err := FALSE;
   S707_LM_DC_FF_PIN.M_Ret_Err := FALSE;
   S707_LM_DC_FF_PIN.LP_Adv := FALSE;
   S707_LM_DC_FF_PIN.LP_Ret := FALSE;
   S707_LM_DC_FF_PIN.Visu_Adv := W#16#0;
   S707_LM_DC_FF_PIN.Visu_Ret := W#16#0;
   S707_LM_DC_FF_PIN.Error_T1.IN := FALSE;
   S707_LM_DC_FF_PIN.Error_T1.PT := T#4S;
   S707_LM_DC_FF_PIN.Error_T1.Q := FALSE;
   S707_LM_DC_FF_PIN.Error_T1.ET := T#0MS;
   S707_LM_DC_FF_PIN.Error_T1.STATE := B#16#0;
   S707_LM_DC_FF_PIN.Error_T1.STIME := T#0MS;
   S707_LM_DC_FF_PIN.Error_T1.ATIME := T#0MS;
   S707_LM_DC_FF_PIN.Error_T2.IN := FALSE;
   S707_LM_DC_FF_PIN.Error_T2.PT := T#4S;
   S707_LM_DC_FF_PIN.Error_T2.Q := FALSE;
   S707_LM_DC_FF_PIN.Error_T2.ET := T#0MS;
   S707_LM_DC_FF_PIN.Error_T2.STATE := B#16#0;
   S707_LM_DC_FF_PIN.Error_T2.STIME := T#0MS;
   S707_LM_DC_FF_PIN.Error_T2.ATIME := T#0MS;
   S707_LM_DC_FF_PIN.CHK_Aux1 := FALSE;
   S707_LM_DC_FF_PIN.CHK_Aux2 := FALSE;
   S707_LM_DC_FF_PIN.Error_T1_DN := FALSE;
   S707_LM_DC_FF_PIN.Error_T2_DN := FALSE;
   S707_LM_DC_FF_PIN.Adv_Memo := FALSE;
   S707_LM_DC_FF_PIN.Visu_Adv_Arr[0] := FALSE;
   S707_LM_DC_FF_PIN.Visu_Adv_Arr[1] := FALSE;
   S707_LM_DC_FF_PIN.Visu_Adv_Arr[2] := FALSE;
   S707_LM_DC_FF_PIN.Visu_Adv_Arr[3] := FALSE;
   S707_LM_DC_FF_PIN.Visu_Adv_Arr[4] := FALSE;
   S707_LM_DC_FF_PIN.Visu_Adv_Arr[5] := FALSE;
   S707_LM_DC_FF_PIN.Visu_Adv_Arr[6] := FALSE;
   S707_LM_DC_FF_PIN.Visu_Adv_Arr[7] := FALSE;
   S707_LM_DC_FF_PIN.Visu_Adv_Arr[8] := FALSE;
   S707_LM_DC_FF_PIN.Visu_Adv_Arr[9] := FALSE;
   S707_LM_DC_FF_PIN.Visu_Adv_Arr[10] := FALSE;
   S707_LM_DC_FF_PIN.Visu_Adv_Arr[11] := FALSE;
   S707_LM_DC_FF_PIN.Visu_Adv_Arr[12] := FALSE;
   S707_LM_DC_FF_PIN.Visu_Adv_Arr[13] := FALSE;
   S707_LM_DC_FF_PIN.Visu_Adv_Arr[14] := FALSE;
   S707_LM_DC_FF_PIN.Visu_Adv_Arr[15] := FALSE;
   S707_LM_DC_FF_PIN.Visu_Ret_Arr[0] := FALSE;
   S707_LM_DC_FF_PIN.Visu_Ret_Arr[1] := FALSE;
   S707_LM_DC_FF_PIN.Visu_Ret_Arr[2] := FALSE;
   S707_LM_DC_FF_PIN.Visu_Ret_Arr[3] := FALSE;
   S707_LM_DC_FF_PIN.Visu_Ret_Arr[4] := FALSE;
   S707_LM_DC_FF_PIN.Visu_Ret_Arr[5] := FALSE;
   S707_LM_DC_FF_PIN.Visu_Ret_Arr[6] := FALSE;
   S707_LM_DC_FF_PIN.Visu_Ret_Arr[7] := FALSE;
   S707_LM_DC_FF_PIN.Visu_Ret_Arr[8] := FALSE;
   S707_LM_DC_FF_PIN.Visu_Ret_Arr[9] := FALSE;
   S707_LM_DC_FF_PIN.Visu_Ret_Arr[10] := FALSE;
   S707_LM_DC_FF_PIN.Visu_Ret_Arr[11] := FALSE;
   S707_LM_DC_FF_PIN.Visu_Ret_Arr[12] := FALSE;
   S707_LM_DC_FF_PIN.Visu_Ret_Arr[13] := FALSE;
   S707_LM_DC_FF_PIN.Visu_Ret_Arr[14] := FALSE;
   S707_LM_DC_FF_PIN.Visu_Ret_Arr[15] := FALSE;
   S707_LM_DC_FF_PIN.BLK_Move_Ret := 0;
   S707_LM_DC_FF_PIN.Enable := FALSE;
   S707_LM_DC_FF_PIN.Adv_End := FALSE;
   S707_LM_DC_FF_PIN.Ret_End := FALSE;
   S707_LM_DC_FF_CLAMP.Enable_Aux := FALSE;
   S707_LM_DC_FF_CLAMP.Adv_Amount := 1;
   S707_LM_DC_FF_CLAMP.Ret_Amount := 1;
   S707_LM_DC_FF_CLAMP.LS_Adv1 := FALSE;
   S707_LM_DC_FF_CLAMP.LS_Ret1 := FALSE;
   S707_LM_DC_FF_CLAMP.LS_Adv2 := FALSE;
   S707_LM_DC_FF_CLAMP.LS_Ret2 := FALSE;
   S707_LM_DC_FF_CLAMP.LS_Adv3 := FALSE;
   S707_LM_DC_FF_CLAMP.LS_Ret3 := FALSE;
   S707_LM_DC_FF_CLAMP.LS_Adv4 := FALSE;
   S707_LM_DC_FF_CLAMP.LS_Ret4 := FALSE;
   S707_LM_DC_FF_CLAMP.SOL_Adv := FALSE;
   S707_LM_DC_FF_CLAMP.SOL_Ret := FALSE;
   S707_LM_DC_FF_CLAMP.M_Ready := TRUE;
   S707_LM_DC_FF_CLAMP.T_CHK1 := T#4S;
   S707_LM_DC_FF_CLAMP.T_CHK2 := T#4S;
   S707_LM_DC_FF_CLAMP.PB_Lamp_CHK := FALSE;
   S707_LM_DC_FF_CLAMP.PB_Error_Rst := FALSE;
   S707_LM_DC_FF_CLAMP.M_FLICK := TRUE;
   S707_LM_DC_FF_CLAMP.M_Adv_Err := FALSE;
   S707_LM_DC_FF_CLAMP.M_Ret_Err := FALSE;
   S707_LM_DC_FF_CLAMP.LP_Adv := FALSE;
   S707_LM_DC_FF_CLAMP.LP_Ret := FALSE;
   S707_LM_DC_FF_CLAMP.Visu_Adv := W#16#0;
   S707_LM_DC_FF_CLAMP.Visu_Ret := W#16#0;
   S707_LM_DC_FF_CLAMP.Error_T1.IN := FALSE;
   S707_LM_DC_FF_CLAMP.Error_T1.PT := T#4S;
   S707_LM_DC_FF_CLAMP.Error_T1.Q := FALSE;
   S707_LM_DC_FF_CLAMP.Error_T1.ET := T#0MS;
   S707_LM_DC_FF_CLAMP.Error_T1.STATE := B#16#0;
   S707_LM_DC_FF_CLAMP.Error_T1.STIME := T#0MS;
   S707_LM_DC_FF_CLAMP.Error_T1.ATIME := T#0MS;
   S707_LM_DC_FF_CLAMP.Error_T2.IN := FALSE;
   S707_LM_DC_FF_CLAMP.Error_T2.PT := T#4S;
   S707_LM_DC_FF_CLAMP.Error_T2.Q := FALSE;
   S707_LM_DC_FF_CLAMP.Error_T2.ET := T#0MS;
   S707_LM_DC_FF_CLAMP.Error_T2.STATE := B#16#0;
   S707_LM_DC_FF_CLAMP.Error_T2.STIME := T#0MS;
   S707_LM_DC_FF_CLAMP.Error_T2.ATIME := T#0MS;
   S707_LM_DC_FF_CLAMP.CHK_Aux1 := FALSE;
   S707_LM_DC_FF_CLAMP.CHK_Aux2 := FALSE;
   S707_LM_DC_FF_CLAMP.Error_T1_DN := FALSE;
   S707_LM_DC_FF_CLAMP.Error_T2_DN := FALSE;
   S707_LM_DC_FF_CLAMP.Adv_Memo := FALSE;
   S707_LM_DC_FF_CLAMP.Visu_Adv_Arr[0] := FALSE;
   S707_LM_DC_FF_CLAMP.Visu_Adv_Arr[1] := FALSE;
   S707_LM_DC_FF_CLAMP.Visu_Adv_Arr[2] := FALSE;
   S707_LM_DC_FF_CLAMP.Visu_Adv_Arr[3] := FALSE;
   S707_LM_DC_FF_CLAMP.Visu_Adv_Arr[4] := FALSE;
   S707_LM_DC_FF_CLAMP.Visu_Adv_Arr[5] := FALSE;
   S707_LM_DC_FF_CLAMP.Visu_Adv_Arr[6] := FALSE;
   S707_LM_DC_FF_CLAMP.Visu_Adv_Arr[7] := FALSE;
   S707_LM_DC_FF_CLAMP.Visu_Adv_Arr[8] := FALSE;
   S707_LM_DC_FF_CLAMP.Visu_Adv_Arr[9] := FALSE;
   S707_LM_DC_FF_CLAMP.Visu_Adv_Arr[10] := FALSE;
   S707_LM_DC_FF_CLAMP.Visu_Adv_Arr[11] := FALSE;
   S707_LM_DC_FF_CLAMP.Visu_Adv_Arr[12] := FALSE;
   S707_LM_DC_FF_CLAMP.Visu_Adv_Arr[13] := FALSE;
   S707_LM_DC_FF_CLAMP.Visu_Adv_Arr[14] := FALSE;
   S707_LM_DC_FF_CLAMP.Visu_Adv_Arr[15] := FALSE;
   S707_LM_DC_FF_CLAMP.Visu_Ret_Arr[0] := FALSE;
   S707_LM_DC_FF_CLAMP.Visu_Ret_Arr[1] := FALSE;
   S707_LM_DC_FF_CLAMP.Visu_Ret_Arr[2] := FALSE;
   S707_LM_DC_FF_CLAMP.Visu_Ret_Arr[3] := FALSE;
   S707_LM_DC_FF_CLAMP.Visu_Ret_Arr[4] := FALSE;
   S707_LM_DC_FF_CLAMP.Visu_Ret_Arr[5] := FALSE;
   S707_LM_DC_FF_CLAMP.Visu_Ret_Arr[6] := FALSE;
   S707_LM_DC_FF_CLAMP.Visu_Ret_Arr[7] := FALSE;
   S707_LM_DC_FF_CLAMP.Visu_Ret_Arr[8] := FALSE;
   S707_LM_DC_FF_CLAMP.Visu_Ret_Arr[9] := FALSE;
   S707_LM_DC_FF_CLAMP.Visu_Ret_Arr[10] := FALSE;
   S707_LM_DC_FF_CLAMP.Visu_Ret_Arr[11] := FALSE;
   S707_LM_DC_FF_CLAMP.Visu_Ret_Arr[12] := FALSE;
   S707_LM_DC_FF_CLAMP.Visu_Ret_Arr[13] := FALSE;
   S707_LM_DC_FF_CLAMP.Visu_Ret_Arr[14] := FALSE;
   S707_LM_DC_FF_CLAMP.Visu_Ret_Arr[15] := FALSE;
   S707_LM_DC_FF_CLAMP.BLK_Move_Ret := 0;
   S707_LM_DC_FF_CLAMP.Enable := FALSE;
   S707_LM_DC_FF_CLAMP.Adv_End := FALSE;
   S707_LM_DC_FF_CLAMP.Ret_End := FALSE;
   S707_LM_DC_2ND_CLAMP6.Enable_Aux := FALSE;
   S707_LM_DC_2ND_CLAMP6.Adv_Amount := 2;
   S707_LM_DC_2ND_CLAMP6.Ret_Amount := 2;
   S707_LM_DC_2ND_CLAMP6.LS_Adv1 := FALSE;
   S707_LM_DC_2ND_CLAMP6.LS_Ret1 := FALSE;
   S707_LM_DC_2ND_CLAMP6.LS_Adv2 := FALSE;
   S707_LM_DC_2ND_CLAMP6.LS_Ret2 := FALSE;
   S707_LM_DC_2ND_CLAMP6.LS_Adv3 := FALSE;
   S707_LM_DC_2ND_CLAMP6.LS_Ret3 := FALSE;
   S707_LM_DC_2ND_CLAMP6.LS_Adv4 := FALSE;
   S707_LM_DC_2ND_CLAMP6.LS_Ret4 := FALSE;
   S707_LM_DC_2ND_CLAMP6.SOL_Adv := FALSE;
   S707_LM_DC_2ND_CLAMP6.SOL_Ret := FALSE;
   S707_LM_DC_2ND_CLAMP6.M_Ready := TRUE;
   S707_LM_DC_2ND_CLAMP6.T_CHK1 := T#4S;
   S707_LM_DC_2ND_CLAMP6.T_CHK2 := T#4S;
   S707_LM_DC_2ND_CLAMP6.PB_Lamp_CHK := FALSE;
   S707_LM_DC_2ND_CLAMP6.PB_Error_Rst := FALSE;
   S707_LM_DC_2ND_CLAMP6.M_FLICK := TRUE;
   S707_LM_DC_2ND_CLAMP6.M_Adv_Err := FALSE;
   S707_LM_DC_2ND_CLAMP6.M_Ret_Err := FALSE;
   S707_LM_DC_2ND_CLAMP6.LP_Adv := FALSE;
   S707_LM_DC_2ND_CLAMP6.LP_Ret := FALSE;
   S707_LM_DC_2ND_CLAMP6.Visu_Adv := W#16#0;
   S707_LM_DC_2ND_CLAMP6.Visu_Ret := W#16#0;
   S707_LM_DC_2ND_CLAMP6.Error_T1.IN := FALSE;
   S707_LM_DC_2ND_CLAMP6.Error_T1.PT := T#4S;
   S707_LM_DC_2ND_CLAMP6.Error_T1.Q := FALSE;
   S707_LM_DC_2ND_CLAMP6.Error_T1.ET := T#0MS;
   S707_LM_DC_2ND_CLAMP6.Error_T1.STATE := B#16#0;
   S707_LM_DC_2ND_CLAMP6.Error_T1.STIME := T#0MS;
   S707_LM_DC_2ND_CLAMP6.Error_T1.ATIME := T#0MS;
   S707_LM_DC_2ND_CLAMP6.Error_T2.IN := FALSE;
   S707_LM_DC_2ND_CLAMP6.Error_T2.PT := T#4S;
   S707_LM_DC_2ND_CLAMP6.Error_T2.Q := FALSE;
   S707_LM_DC_2ND_CLAMP6.Error_T2.ET := T#0MS;
   S707_LM_DC_2ND_CLAMP6.Error_T2.STATE := B#16#0;
   S707_LM_DC_2ND_CLAMP6.Error_T2.STIME := T#0MS;
   S707_LM_DC_2ND_CLAMP6.Error_T2.ATIME := T#0MS;
   S707_LM_DC_2ND_CLAMP6.CHK_Aux1 := FALSE;
   S707_LM_DC_2ND_CLAMP6.CHK_Aux2 := FALSE;
   S707_LM_DC_2ND_CLAMP6.Error_T1_DN := FALSE;
   S707_LM_DC_2ND_CLAMP6.Error_T2_DN := FALSE;
   S707_LM_DC_2ND_CLAMP6.Adv_Memo := TRUE;
   S707_LM_DC_2ND_CLAMP6.Visu_Adv_Arr[0] := FALSE;
   S707_LM_DC_2ND_CLAMP6.Visu_Adv_Arr[1] := FALSE;
   S707_LM_DC_2ND_CLAMP6.Visu_Adv_Arr[2] := FALSE;
   S707_LM_DC_2ND_CLAMP6.Visu_Adv_Arr[3] := FALSE;
   S707_LM_DC_2ND_CLAMP6.Visu_Adv_Arr[4] := FALSE;
   S707_LM_DC_2ND_CLAMP6.Visu_Adv_Arr[5] := FALSE;
   S707_LM_DC_2ND_CLAMP6.Visu_Adv_Arr[6] := FALSE;
   S707_LM_DC_2ND_CLAMP6.Visu_Adv_Arr[7] := FALSE;
   S707_LM_DC_2ND_CLAMP6.Visu_Adv_Arr[8] := FALSE;
   S707_LM_DC_2ND_CLAMP6.Visu_Adv_Arr[9] := FALSE;
   S707_LM_DC_2ND_CLAMP6.Visu_Adv_Arr[10] := FALSE;
   S707_LM_DC_2ND_CLAMP6.Visu_Adv_Arr[11] := FALSE;
   S707_LM_DC_2ND_CLAMP6.Visu_Adv_Arr[12] := FALSE;
   S707_LM_DC_2ND_CLAMP6.Visu_Adv_Arr[13] := FALSE;
   S707_LM_DC_2ND_CLAMP6.Visu_Adv_Arr[14] := FALSE;
   S707_LM_DC_2ND_CLAMP6.Visu_Adv_Arr[15] := FALSE;
   S707_LM_DC_2ND_CLAMP6.Visu_Ret_Arr[0] := FALSE;
   S707_LM_DC_2ND_CLAMP6.Visu_Ret_Arr[1] := FALSE;
   S707_LM_DC_2ND_CLAMP6.Visu_Ret_Arr[2] := FALSE;
   S707_LM_DC_2ND_CLAMP6.Visu_Ret_Arr[3] := FALSE;
   S707_LM_DC_2ND_CLAMP6.Visu_Ret_Arr[4] := FALSE;
   S707_LM_DC_2ND_CLAMP6.Visu_Ret_Arr[5] := FALSE;
   S707_LM_DC_2ND_CLAMP6.Visu_Ret_Arr[6] := FALSE;
   S707_LM_DC_2ND_CLAMP6.Visu_Ret_Arr[7] := FALSE;
   S707_LM_DC_2ND_CLAMP6.Visu_Ret_Arr[8] := FALSE;
   S707_LM_DC_2ND_CLAMP6.Visu_Ret_Arr[9] := FALSE;
   S707_LM_DC_2ND_CLAMP6.Visu_Ret_Arr[10] := FALSE;
   S707_LM_DC_2ND_CLAMP6.Visu_Ret_Arr[11] := FALSE;
   S707_LM_DC_2ND_CLAMP6.Visu_Ret_Arr[12] := FALSE;
   S707_LM_DC_2ND_CLAMP6.Visu_Ret_Arr[13] := FALSE;
   S707_LM_DC_2ND_CLAMP6.Visu_Ret_Arr[14] := FALSE;
   S707_LM_DC_2ND_CLAMP6.Visu_Ret_Arr[15] := FALSE;
   S707_LM_DC_2ND_CLAMP6.BLK_Move_Ret := 0;
   S707_LM_DC_2ND_CLAMP6.Enable := FALSE;
   S707_LM_DC_2ND_CLAMP6.Adv_End := FALSE;
   S707_LM_DC_2ND_CLAMP6.Ret_End := FALSE;
   S707_LM_DC_2ND_CLAMP7.Enable_Aux := FALSE;
   S707_LM_DC_2ND_CLAMP7.Adv_Amount := 1;
   S707_LM_DC_2ND_CLAMP7.Ret_Amount := 1;
   S707_LM_DC_2ND_CLAMP7.LS_Adv1 := FALSE;
